LIN {X 0,Y 144.371,Z 167.125,A -85,B 0,C 180,E1 -25963.188,E2 -25963.188} C_VEL
LIN {X 0,Y 141.893,Z 203.573,A -85,B 0,C 180,E1 -25964.823,E2 -25964.823} C_VEL
LIN {X 0,Y 140.005,Z 216.883,A -85,B 0,C 180,E1 -25965.852,E2 -25965.852} C_VEL
LIN {X 0,Y 137.437,Z 229.509,A -85,B 0,C 180,E1 -25967.347,E2 -25967.347} C_VEL
LIN {X 0,Y 134.351,Z 240.695,A -85,B 0,C 180,E1 -25969.164,E2 -25969.164} C_VEL
LIN {X 0,Y 130.518,Z 252.344,A -85,B 0,C 180,E1 -25971.739,E2 -25971.739} C_VEL
LIN {X 0,Y 127.001,Z 261.752,A -85,B 0,C 180,E1 -25974.475,E2 -25974.475} C_VEL
LIN {X 0,Y 123.23,Z 271.427,A -85,B 0,C 180,E1 -25978.16,E2 -25978.16} C_VEL
LIN {X 0,Y 119.16,Z 280.685,A -85,B 0,C 180,E1 -25982.8,E2 -25982.8} C_VEL
LIN {X 0,Y 116.327,Z 288.174,A -85,B 0,C 180,E1 -25987.814,E2 -25987.814} C_VEL
LIN {X 0,Y 113.848,Z 295.01,A -85,B 0,C 180,E1 -25993.871,E2 -25993.871} C_VEL
LIN {X 0,Y 112.764,Z 299.516,A -85,B 0,C 180,E1 -25999.223,E2 -25999.223} C_VEL
LIN {X 0,Y 112.489,Z 301.887,A -85,B 0,C 180,E1 -26002.822,E2 -26002.822} C_VEL
LIN {X 0,Y 112.546,Z 304.345,A -85,B 0,C 180,E1 -26007.618,E2 -26007.618} C_VEL
LIN {X 0,Y 112.706,Z 305.282,A -85,B 0,C 180,E1 -26010,E2 -26010} C_VEL
LIN {X 0,Y 112.583,Z 306.265,A -85,B 0,C 180,E1 -26013.579,E2 -26013.579} C_VEL
LIN {X 0,Y 112.745,Z 307.033,A -85,B 0,C 180,E1 -26020.778,E2 -26020.778} C_VEL
LIN {X 0,Y 113.483,Z 306.842,A -85,B 0,C 180,E1 -26024.342,E2 -26024.342} C_VEL
LIN {X 0,Y 116.179,Z 305.24,A -85,B 0,C 180,E1 -26031.282,E2 -26031.282} C_VEL
LIN {X 0,Y 120.646,Z 302.091,A -85,B 0,C 180,E1 -26037.777,E2 -26037.777} C_VEL
LIN {X 0,Y 125.355,Z 298.158,A -85,B 0,C 180,E1 -26042.757,E2 -26042.757} C_VEL
LIN {X 0,Y 131.716,Z 292.195,A -85,B 0,C 180,E1 -26047.851,E2 -26047.851} C_VEL
LIN {X 0,Y 137.718,Z 286.001,A -85,B 0,C 180,E1 -26051.561,E2 -26051.561} C_VEL
LIN {X 0,Y 144.339,Z 278.329,A -85,B 0,C 180,E1 -26054.912,E2 -26054.912} C_VEL
LIN {X 0,Y 150.335,Z 270.296,A -85,B 0,C 180,E1 -26057.534,E2 -26057.534} C_VEL
LIN {X 0,Y 151.733,Z 267.559,A -85,B 0,C 180,E1 -26058.493,E2 -26058.493} C_VEL
LIN {X 0,Y 154.006,Z 258.604,A -85,B 0,C 180,E1 -26062.192,E2 -26062.192} C_VEL
LIN {X 0,Y 155.453,Z 255.513,A -85,B 0,C 180,E1 -26062.952,E2 -26062.952} C_VEL
LIN {X 0,Y 160.707,Z 245.469,A -85,B 0,C 180,E1 -26064.539,E2 -26064.539} C_VEL
LIN {X 0,Y 165.609,Z 234.176,A -85,B 0,C 180,E1 -26065.846,E2 -26065.846} C_VEL
LIN {X 0,Y 169.472,Z 222.762,A -85,B 0,C 180,E1 -26066.825,E2 -26066.825} C_VEL
LIN {X 0,Y 172.698,Z 209.662,A -85,B 0,C 180,E1 -26067.587,E2 -26067.587} C_VEL
LIN {X 0,Y 174.718,Z 195.983,A -85,B 0,C 180,E1 -26068.133,E2 -26068.133} C_VEL
LIN {X 0,Y 175.367,Z 187.979,A -85,B 0,C 180,E1 -26068.433,E2 -26068.433} C_VEL
LIN {X 0,Y 172.36,Z 179.063,A -85,B 0,C 180,E1 -26071.315,E2 -26071.315} C_VEL
LIN {X 0,Y 169.405,Z 171.309,A -85,B 0,C 180,E1 -26074.505,E2 -26074.505} C_VEL
LIN {X 0,Y 167.011,Z 165.673,A -85,B 0,C 180,E1 -26077.488,E2 -26077.488} C_VEL
LIN {X 0,Y 165.43,Z 161.949,A -85,B 0,C 180,E1 -26079.827,E2 -26079.827} C_VEL
LIN {X 0,Y 163.63,Z 157.962,A -85,B 0,C 180,E1 -26083.037,E2 -26083.037} C_VEL
LIN {X 0,Y 161.693,Z 154.386,A -85,B 0,C 180,E1 -26087.76,E2 -26087.76} C_VEL
LIN {X 0,Y 161.427,Z 153.804,A -85,B 0,C 180,E1 -26088.701,E2 -26088.701} C_VEL
LIN {X 0,Y 160.411,Z 152.94,A -85,B 0,C 180,E1 -26094.973,E2 -26094.973} C_VEL
LIN {X 0,Y 160.784,Z 152.96,A -85,B 0,C 180,E1 -26099.264,E2 -26099.264} C_VEL
LIN {X 0,Y 161.714,Z 154.006,A -85,B 0,C 180,E1 -26102.958,E2 -26102.958} C_VEL
LIN {X 0,Y 163.636,Z 157.763,A -85,B 0,C 180,E1 -26107.713,E2 -26107.713} C_VEL
LIN {X 0,Y 166.289,Z 162.414,A -85,B 0,C 180,E1 -26112.045,E2 -26112.045} C_VEL
LIN {X 0,Y 168.725,Z 166.769,A -85,B 0,C 180,E1 -26115.128,E2 -26115.128} C_VEL
LIN {X 0,Y 171.773,Z 172.259,A -85,B 0,C 180,E1 -26118.332,E2 -26118.332} C_VEL
LIN {X 0,Y 175.556,Z 179.968,A -85,B 0,C 180,E1 -26121.759,E2 -26121.759} C_VEL
LIN {X 0,Y 175.996,Z 180.975,A -85,B 0,C 180,E1 -26122.132,E2 -26122.132} C_VEL
LIN {X 0,Y 174.142,Z 197.162,A -85,B 0,C 180,E1 -26122.723,E2 -26122.723} C_VEL
LIN {X 0,Y 171.684,Z 209.367,A -85,B 0,C 180,E1 -26123.487,E2 -26123.487} C_VEL
LIN {X 0,Y 168.004,Z 222.113,A -85,B 0,C 180,E1 -26124.651,E2 -26124.651} C_VEL
LIN {X 0,Y 163.378,Z 234.084,A -85,B 0,C 180,E1 -26126.106,E2 -26126.106} C_VEL
LIN {X 0,Y 158.006,Z 244.981,A -85,B 0,C 180,E1 -26127.868,E2 -26127.868} C_VEL
LIN {X 0,Y 152.16,Z 254.847,A -85,B 0,C 180,E1 -26129.999,E2 -26129.999} C_VEL
LIN {X 0,Y 146.008,Z 263.789,A -85,B 0,C 180,E1 -26132.61,E2 -26132.61} C_VEL
LIN {X 0,Y 140.002,Z 271.114,A -85,B 0,C 180,E1 -26135.339,E2 -26135.339} C_VEL
LIN {X 0,Y 134.415,Z 277.166,A -85,B 0,C 180,E1 -26138.345,E2 -26138.345} C_VEL
LIN {X 0,Y 128.196,Z 283.07,A -85,B 0,C 180,E1 -26142.26,E2 -26142.26} C_VEL
LIN {X 0,Y 122.548,Z 287.68,A -85,B 0,C 180,E1 -26146.513,E2 -26146.513} C_VEL
LIN {X 0,Y 118.025,Z 290.872,A -85,B 0,C 180,E1 -26150.724,E2 -26150.724} C_VEL
LIN {X 0,Y 113.464,Z 293.574,A -85,B 0,C 180,E1 -26156.119,E2 -26156.119} C_VEL
LIN {X 0,Y 111.17,Z 294.645,A -85,B 0,C 180,E1 -26159.619,E2 -26159.619} C_VEL
LIN {X 0,Y 107.735,Z 295.552,A -85,B 0,C 180,E1 -26166.958,E2 -26166.958} C_VEL
LIN {X 0,Y 106.539,Z 295.422,A -85,B 0,C 180,E1 -26170.741,E2 -26170.741} C_VEL
LIN {X 0,Y 105.734,Z 294.852,A -85,B 0,C 180,E1 -26174.581,E2 -26174.581} C_VEL
LIN {X 0,Y 105.388,Z 293.878,A -85,B 0,C 180,E1 -26178.46,E2 -26178.46} C_VEL
LIN {X 0,Y 105.77,Z 291.147,A -85,B 0,C 180,E1 -26185.332,E2 -26185.332} C_VEL
LIN {X 0,Y 106.744,Z 287.22,A -85,B 0,C 180,E1 -26191.887,E2 -26191.887} C_VEL
LIN {X 0,Y 108.52,Z 282.62,A -85,B 0,C 180,E1 -26197.442,E2 -26197.442} C_VEL
LIN {X 0,Y 111.491,Z 275.685,A -85,B 0,C 180,E1 -26203.674,E2 -26203.674} C_VEL
LIN {X 0,Y 115.036,Z 268.172,A -85,B 0,C 180,E1 -26208.708,E2 -26208.708} C_VEL
LIN {X 0,Y 118.414,Z 260.521,A -85,B 0,C 180,E1 -26212.693,E2 -26212.693} C_VEL
LIN {X 0,Y 122.438,Z 251.174,A -85,B 0,C 180,E1 -26216.415,E2 -26216.415} C_VEL
LIN {X 0,Y 126.508,Z 240.767,A -85,B 0,C 180,E1 -26219.541,E2 -26219.541} C_VEL
LIN {X 0,Y 130.298,Z 229.231,A -85,B 0,C 180,E1 -26222.184,E2 -26222.184} C_VEL
LIN {X 0,Y 133.405,Z 217.085,A -85,B 0,C 180,E1 -26224.267,E2 -26224.267} C_VEL
LIN {X 0,Y 135.877,Z 203.674,A -85,B 0,C 180,E1 -26225.918,E2 -26225.918} C_VEL
LIN {X 0,Y 137.458,Z 190.843,A -85,B 0,C 180,E1 -26226.941,E2 -26226.941} C_VEL
LIN {X 0,Y 140.322,Z 149.589,A -85,B 0,C 180,E1 -26228.789,E2 -26228.789} C_VEL
LIN {X 0,Y 135.901,Z 140.06,A -85,B 0,C 180,E1 -26231.373,E2 -26231.373} C_VEL
LIN {X 0,Y 131.262,Z 131.57,A -85,B 0,C 180,E1 -26234.301,E2 -26234.301} C_VEL
LIN {X 0,Y 126.15,Z 123.395,A -85,B 0,C 180,E1 -26237.916,E2 -26237.916} C_VEL
LIN {X 0,Y 122.463,Z 118.286,A -85,B 0,C 180,E1 -26240.856,E2 -26240.856} C_VEL
LIN {X 0,Y 120.026,Z 114.83,A -85,B 0,C 180,E1 -26243.049,E2 -26243.049} C_VEL
LIN {X 0,Y 117.541,Z 111.714,A -85,B 0,C 180,E1 -26245.488,E2 -26245.488} C_VEL
LIN {X 0,Y 116.829,Z 110.266,A -85,B 0,C 180,E1 -26246.312,E2 -26246.312} C_VEL
LIN {X 0,Y 114.195,Z 107.957,A -85,B 0,C 180,E1 -26249.228,E2 -26249.228} C_VEL
LIN {X 0,Y 112.545,Z 104.889,A -85,B 0,C 180,E1 -26251.566,E2 -26251.566} C_VEL
LIN {X 0,Y 109.927,Z 103.24,A -85,B 0,C 180,E1 -26255.365,E2 -26255.365} C_VEL
LIN {X 0,Y 108.274,Z 100.512,A -85,B 0,C 180,E1 -26258.711,E2 -26258.711} C_VEL
LIN {X 0,Y 107.884,Z 99.025,A -85,B 0,C 180,E1 -26260.001,E2 -26260.001} C_VEL
LIN {X 0,Y 108.177,Z 98.985,A -85,B 0,C 180,E1 -26267.039,E2 -26267.039} C_VEL
LIN {X 0,Y 108.305,Z 98.962,A -85,B 0,C 180,E1 -26272.543,E2 -26272.543} C_VEL
LIN {X 0,Y 108.92,Z 98.908,A -85,B 0,C 180,E1 -26280,E2 -26280} C_VEL
LIN {X 0,Y 108.27,Z 99.01,A -85,B 0,C 180,E1 -26290.165,E2 -26290.165} C_VEL
LIN {X 0,Y 108.973,Z 101.41,A -85,B 0,C 180,E1 -26291.986,E2 -26291.986} C_VEL
LIN {X 0,Y 110.885,Z 103.905,A -85,B 0,C 180,E1 -26295.392,E2 -26295.392} C_VEL
LIN {X 0,Y 112.887,Z 105.114,A -85,B 0,C 180,E1 -26298.137,E2 -26298.137} C_VEL
LIN {X 0,Y 114.533,Z 108.231,A -85,B 0,C 180,E1 -26300.426,E2 -26300.426} C_VEL
LIN {X 0,Y 117.047,Z 110.636,A -85,B 0,C 180,E1 -26303.189,E2 -26303.189} C_VEL
LIN {X 0,Y 119.289,Z 114.04,A -85,B 0,C 180,E1 -26305.52,E2 -26305.52} C_VEL
LIN {X 0,Y 120.811,Z 115.735,A -85,B 0,C 180,E1 -26306.908,E2 -26306.908} C_VEL
LIN {X 0,Y 124.326,Z 120.81,A -85,B 0,C 180,E1 -26309.92,E2 -26309.92} C_VEL
LIN {X 0,Y 128.722,Z 127.364,A -85,B 0,C 180,E1 -26313.209,E2 -26313.209} C_VEL
LIN {X 0,Y 132.754,Z 136.18,A -85,B 0,C 180,E1 -26316.083,E2 -26316.083} C_VEL
LIN {X 0,Y 136.377,Z 145.541,A -85,B 0,C 180,E1 -26318.505,E2 -26318.505} C_VEL
LIN {X 0,Y 138.617,Z 152.722,A -85,B 0,C 180,E1 -26319.99,E2 -26319.99} C_VEL
LIN {X 0,Y 139.093,Z 168.621,A -85,B 0,C 180,E1 -26321.313,E2 -26321.313} C_VEL
LIN {X 0,Y 136.557,Z 203.434,A -85,B 0,C 180,E1 -26322.9,E2 -26322.9} C_VEL
LIN {X 0,Y 134.553,Z 216.833,A -85,B 0,C 180,E1 -26323.959,E2 -26323.959} C_VEL
LIN {X 0,Y 132.023,Z 228.822,A -85,B 0,C 180,E1 -26325.41,E2 -26325.41} C_VEL
LIN {X 0,Y 128.519,Z 240.886,A -85,B 0,C 180,E1 -26327.411,E2 -26327.411} C_VEL
LIN {X 0,Y 124.509,Z 252.43,A -85,B 0,C 180,E1 -26330.053,E2 -26330.053} C_VEL
LIN {X 0,Y 120.805,Z 261.755,A -85,B 0,C 180,E1 -26332.873,E2 -26332.873} C_VEL
LIN {X 0,Y 117.188,Z 270.462,A -85,B 0,C 180,E1 -26336.306,E2 -26336.306} C_VEL
LIN {X 0,Y 114.298,Z 276.8,A -85,B 0,C 180,E1 -26339.411,E2 -26339.411} C_VEL
LIN {X 0,Y 112.238,Z 281.288,A -85,B 0,C 180,E1 -26342.026,E2 -26342.026} C_VEL
LIN {X 0,Y 109.277,Z 288.558,A -85,B 0,C 180,E1 -26347.301,E2 -26347.301} C_VEL
LIN {X 0,Y 106.988,Z 294.362,A -85,B 0,C 180,E1 -26352.806,E2 -26352.806} C_VEL
LIN {X 0,Y 105.766,Z 298.93,A -85,B 0,C 180,E1 -26358.501,E2 -26358.501} C_VEL
LIN {X 0,Y 105.42,Z 301.33,A -85,B 0,C 180,E1 -26362.337,E2 -26362.337} C_VEL
LIN {X 0,Y 105.48,Z 304.085,A -85,B 0,C 180,E1 -26368.092,E2 -26368.092} C_VEL
LIN {X 0,Y 105.608,Z 304.802,A -85,B 0,C 180,E1 -26370,E2 -26370} C_VEL
LIN {X 0,Y 105.495,Z 305.815,A -85,B 0,C 180,E1 -26373.82,E2 -26373.82} C_VEL
LIN {X 0,Y 105.759,Z 306.634,A -85,B 0,C 180,E1 -26381.499,E2 -26381.499} C_VEL
LIN {X 0,Y 106.57,Z 306.478,A -85,B 0,C 180,E1 -26385.295,E2 -26385.295} C_VEL
LIN {X 0,Y 107.8,Z 305.906,A -85,B 0,C 180,E1 -26389.024,E2 -26389.024} C_VEL
LIN {X 0,Y 111.781,Z 303.597,A -85,B 0,C 180,E1 -26396.111,E2 -26396.111} C_VEL
LIN {X 0,Y 115.858,Z 300.796,A -85,B 0,C 180,E1 -26401.039,E2 -26401.039} C_VEL
LIN {X 0,Y 120.643,Z 296.997,A -85,B 0,C 180,E1 -26405.63,E2 -26405.63} C_VEL
LIN {X 0,Y 126.173,Z 292.108,A -85,B 0,C 180,E1 -26409.834,E2 -26409.834} C_VEL
LIN {X 0,Y 132.494,Z 285.984,A -85,B 0,C 180,E1 -26413.596,E2 -26413.596} C_VEL
LIN {X 0,Y 139.397,Z 278.403,A -85,B 0,C 180,E1 -26416.975,E2 -26416.975} C_VEL
LIN {X 0,Y 145.489,Z 270.684,A -85,B 0,C 180,E1 -26419.537,E2 -26419.537} C_VEL
LIN {X 0,Y 152.555,Z 260.232,A -85,B 0,C 180,E1 -26422.086,E2 -26422.086} C_VEL
LIN {X 0,Y 155.453,Z 255.513,A -85,B 0,C 180,E1 -26422.952,E2 -26422.952} C_VEL
LIN {X 0,Y 157.735,Z 250.79,A -85,B 0,C 180,E1 -26423.931,E2 -26423.931} C_VEL
LIN {X 0,Y 160.132,Z 242.902,A -85,B 0,C 180,E1 -26425.914,E2 -26425.914} C_VEL
LIN {X 0,Y 162.217,Z 234.678,A -85,B 0,C 180,E1 -26427.726,E2 -26427.726} C_VEL
LIN {X 0,Y 163.888,Z 229.337,A -85,B 0,C 180,E1 -26428.437,E2 -26428.437} C_VEL
LIN {X 0,Y 167.933,Z 216.125,A -85,B 0,C 180,E1 -26429.373,E2 -26429.373} C_VEL
LIN {X 0,Y 170.635,Z 203.005,A -85,B 0,C 180,E1 -26429.982,E2 -26429.982} C_VEL
LIN {X 0,Y 171.993,Z 190.995,A -85,B 0,C 180,E1 -26430.412,E2 -26430.412} C_VEL
LIN {X 0,Y 169.101,Z 182.07,A -85,B 0,C 180,E1 -26433.545,E2 -26433.545} C_VEL
LIN {X 0,Y 166.5,Z 174.975,A -85,B 0,C 180,E1 -26436.771,E2 -26436.771} C_VEL
LIN {X 0,Y 163.949,Z 168.443,A -85,B 0,C 180,E1 -26440.657,E2 -26440.657} C_VEL
LIN {X 0,Y 162.391,Z 164.745,A -85,B 0,C 180,E1 -26443.661,E2 -26443.661} C_VEL
LIN {X 0,Y 160.595,Z 161.098,A -85,B 0,C 180,E1 -26448.479,E2 -26448.479} C_VEL
LIN {X 0,Y 159.74,Z 160.172,A -85,B 0,C 180,E1 -26452.415,E2 -26452.415} C_VEL
LIN {X 0,Y 159.823,Z 159.956,A -85,B 0,C 180,E1 -26458.74,E2 -26458.74} C_VEL
LIN {X 0,Y 160.683,Z 160.956,A -85,B 0,C 180,E1 -26462.507,E2 -26462.507} C_VEL
LIN {X 0,Y 162.454,Z 164.606,A -85,B 0,C 180,E1 -26467.196,E2 -26467.196} C_VEL
LIN {X 0,Y 164.873,Z 169.197,A -85,B 0,C 180,E1 -26471.407,E2 -26471.407} C_VEL
LIN {X 0,Y 167.262,Z 173.689,A -85,B 0,C 180,E1 -26474.602,E2 -26474.602} C_VEL
LIN {X 0,Y 169.943,Z 178.878,A -85,B 0,C 180,E1 -26477.583,E2 -26477.583} C_VEL
LIN {X 0,Y 172.573,Z 184.626,A -85,B 0,C 180,E1 -26480.168,E2 -26480.168} C_VEL
LIN {X 0,Y 170.743,Z 198.637,A -85,B 0,C 180,E1 -26480.681,E2 -26480.681} C_VEL
LIN {X 0,Y 167.955,Z 211.364,A -85,B 0,C 180,E1 -26481.495,E2 -26481.495} C_VEL
LIN {X 0,Y 164.109,Z 223.915,A -85,B 0,C 180,E1 -26482.67,E2 -26482.67} C_VEL
LIN {X 0,Y 159.627,Z 234.869,A -85,B 0,C 180,E1 -26483.995,E2 -26483.995} C_VEL
LIN {X 0,Y 154.062,Z 245.674,A -85,B 0,C 180,E1 -26485.715,E2 -26485.715} C_VEL
LIN {X 0,Y 147.811,Z 255.787,A -85,B 0,C 180,E1 -26487.897,E2 -26487.897} C_VEL
LIN {X 0,Y 140.957,Z 265.198,A -85,B 0,C 180,E1 -26490.675,E2 -26490.675} C_VEL
LIN {X 0,Y 133.525,Z 273.587,A -85,B 0,C 180,E1 -26494.005,E2 -26494.005} C_VEL
LIN {X 0,Y 127.127,Z 279.857,A -85,B 0,C 180,E1 -26497.453,E2 -26497.453} C_VEL
LIN {X 0,Y 121.328,Z 284.805,A -85,B 0,C 180,E1 -26501.146,E2 -26501.146} C_VEL
LIN {X 0,Y 115.517,Z 289.09,A -85,B 0,C 180,E1 -26505.601,E2 -26505.601} C_VEL
LIN {X 0,Y 110.436,Z 292.27,A -85,B 0,C 180,E1 -26510.477,E2 -26510.477} C_VEL
LIN {X 0,Y 107.498,Z 293.83,A -85,B 0,C 180,E1 -26513.956,E2 -26513.956} C_VEL
LIN {X 0,Y 104.965,Z 294.961,A -85,B 0,C 180,E1 -26517.612,E2 -26517.612} C_VEL
LIN {X 0,Y 101.108,Z 295.929,A -85,B 0,C 180,E1 -26525.351,E2 -26525.351} C_VEL
LIN {X 0,Y 99.757,Z 295.83,A -85,B 0,C 180,E1 -26529.375,E2 -26529.375} C_VEL
LIN {X 0,Y 98.793,Z 295.319,A -85,B 0,C 180,E1 -26533.468,E2 -26533.468} C_VEL
LIN {X 0,Y 98.339,Z 294.374,A -85,B 0,C 180,E1 -26537.62,E2 -26537.62} C_VEL
LIN {X 0,Y 98.695,Z 291.476,A -85,B 0,C 180,E1 -26545.503,E2 -26545.503} C_VEL
LIN {X 0,Y 99.646,Z 287.846,A -85,B 0,C 180,E1 -26552.021,E2 -26552.021} C_VEL
LIN {X 0,Y 101.497,Z 283.321,A -85,B 0,C 180,E1 -26557.961,E2 -26557.961} C_VEL
LIN {X 0,Y 104.605,Z 276.484,A -85,B 0,C 180,E1 -26564.593,E2 -26564.593} C_VEL
LIN {X 0,Y 108.356,Z 269.056,A -85,B 0,C 180,E1 -26569.909,E2 -26569.909} C_VEL
LIN {X 0,Y 111.934,Z 261.504,A -85,B 0,C 180,E1 -26574.087,E2 -26574.087} C_VEL
LIN {X 0,Y 116.138,Z 252.336,A -85,B 0,C 180,E1 -26577.969,E2 -26577.969} C_VEL
LIN {X 0,Y 120.38,Z 242.112,A -85,B 0,C 180,E1 -26581.208,E2 -26581.208} C_VEL
LIN {X 0,Y 124.385,Z 230.781,A -85,B 0,C 180,E1 -26583.915,E2 -26583.915} C_VEL
LIN {X 0,Y 127.667,Z 219.064,A -85,B 0,C 180,E1 -26586.04,E2 -26586.04} C_VEL
LIN {X 0,Y 130.268,Z 206.292,A -85,B 0,C 180,E1 -26587.726,E2 -26587.726} C_VEL
LIN {X 0,Y 132.135,Z 192.787,A -85,B 0,C 180,E1 -26588.898,E2 -26588.898} C_VEL
LIN {X 0,Y 135.181,Z 151.945,A -85,B 0,C 180,E1 -26590.79,E2 -26590.79} C_VEL
LIN {X 0,Y 131.121,Z 143.155,A -85,B 0,C 180,E1 -26593.409,E2 -26593.409} C_VEL
LIN {X 0,Y 126.794,Z 135.129,A -85,B 0,C 180,E1 -26596.443,E2 -26596.443} C_VEL
LIN {X 0,Y 122.314,Z 127.979,A -85,B 0,C 180,E1 -26599.955,E2 -26599.955} C_VEL
LIN {X 0,Y 119.3,Z 123.587,A -85,B 0,C 180,E1 -26602.625,E2 -26602.625} C_VEL
LIN {X 0,Y 117.486,Z 120.881,A -85,B 0,C 180,E1 -26604.413,E2 -26604.413} C_VEL
LIN {X 0,Y 114.951,Z 117.413,A -85,B 0,C 180,E1 -26607.142,E2 -26607.142} C_VEL
LIN {X 0,Y 114.18,Z 116.359,A -85,B 0,C 180,E1 -26608.049,E2 -26608.049} C_VEL
LIN {X 0,Y 111.847,Z 113.755,A -85,B 0,C 180,E1 -26610.978,E2 -26610.978} C_VEL
LIN {X 0,Y 110.772,Z 111.622,A -85,B 0,C 180,E1 -26612.655,E2 -26612.655} C_VEL
LIN {X 0,Y 108.173,Z 109.622,A -85,B 0,C 180,E1 -26616.819,E2 -26616.819} C_VEL
LIN {X 0,Y 106.685,Z 106.794,A -85,B 0,C 180,E1 -26620.269,E2 -26620.269} C_VEL
LIN {X 0,Y 106.364,Z 105.942,A -85,B 0,C 180,E1 -26621.21,E2 -26621.21} C_VEL
LIN {X 0,Y 103.763,Z 104.443,A -85,B 0,C 180,E1 -26632.215,E2 -26632.215} C_VEL
LIN {X 0,Y 104.224,Z 104.336,A -85,B 0,C 180,E1 -26640.483,E2 -26640.483} C_VEL
LIN {X 0,Y 106.798,Z 106.137,A -85,B 0,C 180,E1 -26649.042,E2 -26649.042} C_VEL
LIN {X 0,Y 108.097,Z 109.161,A -85,B 0,C 180,E1 -26652.199,E2 -26652.199} C_VEL
LIN {X 0,Y 110.242,Z 111.258,A -85,B 0,C 180,E1 -26655.839,E2 -26655.839} C_VEL
LIN {X 0,Y 111.072,Z 111.982,A -85,B 0,C 180,E1 -26657.046,E2 -26657.046} C_VEL
LIN {X 0,Y 112.976,Z 115.135,A -85,B 0,C 180,E1 -26659.771,E2 -26659.771} C_VEL
LIN {X 0,Y 114.795,Z 116.994,A -85,B 0,C 180,E1 -26661.906,E2 -26661.906} C_VEL
LIN {X 0,Y 117.423,Z 120.762,A -85,B 0,C 180,E1 -26664.77,E2 -26664.77} C_VEL
LIN {X 0,Y 121.111,Z 126.062,A -85,B 0,C 180,E1 -26668.249,E2 -26668.249} C_VEL
LIN {X 0,Y 125.451,Z 132.911,A -85,B 0,C 180,E1 -26671.801,E2 -26671.801} C_VEL
LIN {X 0,Y 129.768,Z 143.114,A -85,B 0,C 180,E1 -26675.14,E2 -26675.14} C_VEL
LIN {X 0,Y 133.589,Z 154.367,A -85,B 0,C 180,E1 -26677.923,E2 -26677.923} C_VEL
LIN {X 0,Y 134.045,Z 168.599,A -85,B 0,C 180,E1 -26679.218,E2 -26679.218} C_VEL
LIN {X 0,Y 131.514,Z 202.469,A -85,B 0,C 180,E1 -26680.791,E2 -26680.791} C_VEL
LIN {X 0,Y 129.435,Z 215.975,A -85,B 0,C 180,E1 -26681.849,E2 -26681.849} C_VEL
LIN {X 0,Y 126.773,Z 228.088,A -85,B 0,C 180,E1 -26683.312,E2 -26683.312} C_VEL
LIN {X 0,Y 123.382,Z 239.46,A -85,B 0,C 180,E1 -26685.178,E2 -26685.178} C_VEL
LIN {X 0,Y 120.222,Z 248.562,A -85,B 0,C 180,E1 -26687.188,E2 -26687.188} C_VEL
LIN {X 0,Y 115.58,Z 259.567,A -85,B 0,C 180,E1 -26690.322,E2 -26690.322} C_VEL
LIN {X 0,Y 112.112,Z 267.679,A -85,B 0,C 180,E1 -26693.449,E2 -26693.449} C_VEL
LIN {X 0,Y 108.084,Z 276.238,A -85,B 0,C 180,E1 -26697.669,E2 -26697.669} C_VEL
LIN {X 0,Y 105.753,Z 280.839,A -85,B 0,C 180,E1 -26700.45,E2 -26700.45} C_VEL
LIN {X 0,Y 102.709,Z 287.81,A -85,B 0,C 180,E1 -26705.76,E2 -26705.76} C_VEL
LIN {X 0,Y 100.181,Z 293.703,A -85,B 0,C 180,E1 -26711.597,E2 -26711.597} C_VEL
LIN {X 0,Y 98.759,Z 298.338,A -85,B 0,C 180,E1 -26717.673,E2 -26717.673} C_VEL
LIN {X 0,Y 98.347,Z 300.772,A -85,B 0,C 180,E1 -26721.783,E2 -26721.783} C_VEL
LIN {X 0,Y 98.431,Z 303.75,A -85,B 0,C 180,E1 -26728.416,E2 -26728.416} C_VEL
LIN {X 0,Y 98.445,Z 304.824,A -85,B 0,C 180,E1 -26731.86,E2 -26731.86} C_VEL
LIN {X 0,Y 98.349,Z 305.988,A -85,B 0,C 180,E1 -26738.217,E2 -26738.217} C_VEL
LIN {X 0,Y 99.7,Z 306.104,A -85,B 0,C 180,E1 -26746.377,E2 -26746.377} C_VEL
LIN {X 0,Y 101.079,Z 305.584,A -85,B 0,C 180,E1 -26750.343,E2 -26750.343} C_VEL
LIN {X 0,Y 105.418,Z 303.33,A -85,B 0,C 180,E1 -26757.819,E2 -26757.819} C_VEL
LIN {X 0,Y 109.803,Z 300.585,A -85,B 0,C 180,E1 -26762.96,E2 -26762.96} C_VEL
LIN {X 0,Y 114.932,Z 296.846,A -85,B 0,C 180,E1 -26767.698,E2 -26767.698} C_VEL
LIN {X 0,Y 120.806,Z 292.021,A -85,B 0,C 180,E1 -26771.992,E2 -26771.992} C_VEL
LIN {X 0,Y 127.445,Z 285.967,A -85,B 0,C 180,E1 -26775.798,E2 -26775.798} C_VEL
LIN {X 0,Y 134.65,Z 278.465,A -85,B 0,C 180,E1 -26779.185,E2 -26779.185} C_VEL
LIN {X 0,Y 140.99,Z 270.837,A -85,B 0,C 180,E1 -26781.73,E2 -26781.73} C_VEL
LIN {X 0,Y 147.612,Z 261.615,A -85,B 0,C 180,E1 -26784.037,E2 -26784.037} C_VEL
LIN {X 0,Y 153.194,Z 252.645,A -85,B 0,C 180,E1 -26785.668,E2 -26785.668} C_VEL
LIN {X 0,Y 158.865,Z 241.602,A -85,B 0,C 180,E1 -26787.197,E2 -26787.197} C_VEL
LIN {X 0,Y 163.888,Z 229.337,A -85,B 0,C 180,E1 -26788.437,E2 -26788.437} C_VEL
LIN {X 0,Y 164.842,Z 225.742,A -85,B 0,C 180,E1 -26788.951,E2 -26788.951} C_VEL
LIN {X 0,Y 165.341,Z 220.112,A -85,B 0,C 180,E1 -26790.25,E2 -26790.25} C_VEL
LIN {X 0,Y 165.642,Z 214.358,A -85,B 0,C 180,E1 -26791.465,E2 -26791.465} C_VEL
LIN {X 0,Y 166.219,Z 210.576,A -85,B 0,C 180,E1 -26791.843,E2 -26791.843} C_VEL
LIN {X 0,Y 168.391,Z 197.785,A -85,B 0,C 180,E1 -26792.355,E2 -26792.355} C_VEL
LIN {X 0,Y 168.795,Z 194.083,A -85,B 0,C 180,E1 -26792.488,E2 -26792.488} C_VEL
LIN {X 0,Y 166.577,Z 186.757,A -85,B 0,C 180,E1 -26795.211,E2 -26795.211} C_VEL
LIN {X 0,Y 164.431,Z 180.436,A -85,B 0,C 180,E1 -26798.203,E2 -26798.203} C_VEL
LIN {X 0,Y 162.329,Z 174.605,A -85,B 0,C 180,E1 -26801.811,E2 -26801.811} C_VEL
LIN {X 0,Y 161.081,Z 171.394,A -85,B 0,C 180,E1 -26804.49,E2 -26804.49} C_VEL
LIN {X 0,Y 159.523,Z 167.814,A -85,B 0,C 180,E1 -26809.208,E2 -26809.208} C_VEL
LIN {X 0,Y 158.671,Z 167.039,A -85,B 0,C 180,E1 -26814.917,E2 -26814.917} C_VEL
LIN {X 0,Y 158.949,Z 167.008,A -85,B 0,C 180,E1 -26818.733,E2 -26818.733} C_VEL
LIN {X 0,Y 159.657,Z 167.938,A -85,B 0,C 180,E1 -26822.049,E2 -26822.049} C_VEL
LIN {X 0,Y 161.587,Z 172.161,A -85,B 0,C 180,E1 -26827.34,E2 -26827.34} C_VEL
LIN {X 0,Y 163.624,Z 176.25,A -85,B 0,C 180,E1 -26830.988,E2 -26830.988} C_VEL
LIN {X 0,Y 166.198,Z 181.331,A -85,B 0,C 180,E1 -26834.541,E2 -26834.541} C_VEL
LIN {X 0,Y 169.03,Z 187.503,A -85,B 0,C 180,E1 -26837.779,E2 -26837.779} C_VEL
LIN {X 0,Y 169.273,Z 188.079,A -85,B 0,C 180,E1 -26838.046,E2 -26838.046} C_VEL
LIN {X 0,Y 167.298,Z 201.388,A -85,B 0,C 180,E1 -26838.629,E2 -26838.629} C_VEL
LIN {X 0,Y 164.063,Z 214.777,A -85,B 0,C 180,E1 -26839.537,E2 -26839.537} C_VEL
LIN {X 0,Y 159.658,Z 227.45,A -85,B 0,C 180,E1 -26840.766,E2 -26840.766} C_VEL
LIN {X 0,Y 154.646,Z 238.535,A -85,B 0,C 180,E1 -26842.186,E2 -26842.186} C_VEL
LIN {X 0,Y 148.221,Z 249.87,A -85,B 0,C 180,E1 -26844.111,E2 -26844.111} C_VEL
LIN {X 0,Y 141.366,Z 259.881,A -85,B 0,C 180,E1 -26846.508,E2 -26846.508} C_VEL
LIN {X 0,Y 134.741,Z 268.036,A -85,B 0,C 180,E1 -26849.112,E2 -26849.112} C_VEL
LIN {X 0,Y 127.136,Z 275.978,A -85,B 0,C 180,E1 -26852.54,E2 -26852.54} C_VEL
LIN {X 0,Y 121.177,Z 281.326,A -85,B 0,C 180,E1 -26855.711,E2 -26855.711} C_VEL
LIN {X 0,Y 114.52,Z 286.499,A -85,B 0,C 180,E1 -26859.904,E2 -26859.904} C_VEL
LIN {X 0,Y 108.516,Z 290.472,A -85,B 0,C 180,E1 -26864.569,E2 -26864.569} C_VEL
LIN {X 0,Y 104.933,Z 292.493,A -85,B 0,C 180,E1 -26867.951,E2 -26867.951} C_VEL
LIN {X 0,Y 101.712,Z 294.085,A -85,B 0,C 180,E1 -26871.547,E2 -26871.547} C_VEL
LIN {X 0,Y 98.896,Z 295.264,A -85,B 0,C 180,E1 -26875.353,E2 -26875.353} C_VEL
LIN {X 0,Y 94.948,Z 296.281,A -85,B 0,C 180,E1 -26882.652,E2 -26882.652} C_VEL
LIN {X 0,Y 93.026,Z 296.236,A -85,B 0,C 180,E1 -26887.806,E2 -26887.806} C_VEL
LIN {X 0,Y 91.895,Z 295.777,A -85,B 0,C 180,E1 -26892.187,E2 -26892.187} C_VEL
LIN {X 0,Y 91.312,Z 294.87,A -85,B 0,C 180,E1 -26896.65,E2 -26896.65} C_VEL
LIN {X 0,Y 91.199,Z 293.561,A -85,B 0,C 180,E1 -26901.134,E2 -26901.134} C_VEL
LIN {X 0,Y 91.729,Z 291.241,A -85,B 0,C 180,E1 -26906.937,E2 -26906.937} C_VEL
LIN {X 0,Y 93.041,Z 287.092,A -85,B 0,C 180,E1 -26914.332,E2 -26914.332} C_VEL
LIN {X 0,Y 95.289,Z 282.25,A -85,B 0,C 180,E1 -26920.626,E2 -26920.626} C_VEL
LIN {X 0,Y 98.352,Z 276.165,A -85,B 0,C 180,E1 -26926.609,E2 -26926.609} C_VEL
LIN {X 0,Y 102.453,Z 268.587,A -85,B 0,C 180,E1 -26932.166,E2 -26932.166} C_VEL
LIN {X 0,Y 106.342,Z 260.855,A -85,B 0,C 180,E1 -26936.494,E2 -26936.494} C_VEL
LIN {X 0,Y 110.898,Z 251.386,A -85,B 0,C 180,E1 -26940.464,E2 -26940.464} C_VEL
LIN {X 0,Y 115.455,Z 240.862,A -85,B 0,C 180,E1 -26943.743,E2 -26943.743} C_VEL
LIN {X 0,Y 119.658,Z 229.161,A -85,B 0,C 180,E1 -26946.491,E2 -26946.491} C_VEL
LIN {X 0,Y 123.108,Z 216.69,A -85,B 0,C 180,E1 -26948.639,E2 -26948.639} C_VEL
LIN {X 0,Y 125.762,Z 203.369,A -85,B 0,C 180,E1 -26950.29,E2 -26950.29} C_VEL
LIN {X 0,Y 127.443,Z 190.212,A -85,B 0,C 180,E1 -26951.309,E2 -26951.309} C_VEL
LIN {X 0,Y 130.186,Z 154.306,A -85,B 0,C 180,E1 -26952.959,E2 -26952.959} C_VEL
LIN {X 0,Y 125.815,Z 144.858,A -85,B 0,C 180,E1 -26956.125,E2 -26956.125} C_VEL
LIN {X 0,Y 121.458,Z 136.997,A -85,B 0,C 180,E1 -26959.615,E2 -26959.615} C_VEL
LIN {X 0,Y 116.909,Z 129.812,A -85,B 0,C 180,E1 -26963.825,E2 -26963.825} C_VEL
LIN {X 0,Y 114.851,Z 126.777,A -85,B 0,C 180,E1 -26966.003,E2 -26966.003} C_VEL
LIN {X 0,Y 112.047,Z 122.723,A -85,B 0,C 180,E1 -26969.373,E2 -26969.373} C_VEL
LIN {X 0,Y 109.654,Z 119.617,A -85,B 0,C 180,E1 -26972.725,E2 -26972.725} C_VEL
LIN {X 0,Y 108.959,Z 118.287,A -85,B 0,C 180,E1 -26973.902,E2 -26973.902} C_VEL
LIN {X 0,Y 106.332,Z 115.729,A -85,B 0,C 180,E1 -26978.684,E2 -26978.684} C_VEL
LIN {X 0,Y 105.144,Z 112.948,A -85,B 0,C 180,E1 -26981.993,E2 -26981.993} C_VEL
LIN {X 0,Y 102.896,Z 111.498,A -85,B 0,C 180,E1 -26992.149,E2 -26992.149} C_VEL
LIN {X 0,Y 103.344,Z 111.429,A -85,B 0,C 180,E1 -27000.488,E2 -27000.488} C_VEL
LIN {X 0,Y 105.416,Z 112.981,A -85,B 0,C 180,E1 -27007.918,E2 -27007.918} C_VEL
LIN {X 0,Y 107.055,Z 116.435,A -85,B 0,C 180,E1 -27012.031,E2 -27012.031} C_VEL
LIN {X 0,Y 109.283,Z 118.644,A -85,B 0,C 180,E1 -27015.862,E2 -27015.862} C_VEL
LIN {X 0,Y 111.484,Z 122.03,A -85,B 0,C 180,E1 -27019.153,E2 -27019.153} C_VEL
LIN {X 0,Y 112.723,Z 123.52,A -85,B 0,C 180,E1 -27020.723,E2 -27020.723} C_VEL
LIN {X 0,Y 116.124,Z 128.548,A -85,B 0,C 180,E1 -27024.607,E2 -27024.607} C_VEL
LIN {X 0,Y 120.265,Z 134.93,A -85,B 0,C 180,E1 -27028.585,E2 -27028.585} C_VEL
LIN {X 0,Y 122.466,Z 138.993,A -85,B 0,C 180,E1 -27030.506,E2 -27030.506} C_VEL
LIN {X 0,Y 126.207,Z 148.587,A -85,B 0,C 180,E1 -27033.682,E2 -27033.682} C_VEL
LIN {X 0,Y 128.936,Z 157.158,A -85,B 0,C 180,E1 -27035.891,E2 -27035.891} C_VEL
LIN {X 0,Y 129.115,Z 169.756,A -85,B 0,C 180,E1 -27037.024,E2 -27037.024} C_VEL
LIN {X 0,Y 126.425,Z 202.871,A -85,B 0,C 180,E1 -27038.579,E2 -27038.579} C_VEL
LIN {X 0,Y 124.157,Z 216.618,A -85,B 0,C 180,E1 -27039.691,E2 -27039.691} C_VEL
LIN {X 0,Y 121.398,Z 228.459,A -85,B 0,C 180,E1 -27041.183,E2 -27041.183} C_VEL
LIN {X 0,Y 117.851,Z 239.618,A -85,B 0,C 180,E1 -27043.069,E2 -27043.069} C_VEL
LIN {X 0,Y 113.997,Z 249.962,A -85,B 0,C 180,E1 -27045.469,E2 -27045.469} C_VEL
LIN {X 0,Y 109.175,Z 260.631,A -85,B 0,C 180,E1 -27048.712,E2 -27048.712} C_VEL
LIN {X 0,Y 104.71,Z 270.314,A -85,B 0,C 180,E1 -27052.837,E2 -27052.837} C_VEL
LIN {X 0,Y 100.328,Z 278.456,A -85,B 0,C 180,E1 -27057.357,E2 -27057.357} C_VEL
LIN {X 0,Y 96.727,Z 285.909,A -85,B 0,C 180,E1 -27062.991,E2 -27062.991} C_VEL
LIN {X 0,Y 94.23,Z 291.18,A -85,B 0,C 180,E1 -27068.104,E2 -27068.104} C_VEL
LIN {X 0,Y 92.207,Z 296.274,A -85,B 0,C 180,E1 -27074.527,E2 -27074.527} C_VEL
LIN {X 0,Y 91.309,Z 300.21,A -85,B 0,C 180,E1 -27081.144,E2 -27081.144} C_VEL
LIN {X 0,Y 91.379,Z 303.481,A -85,B 0,C 180,E1 -27089.009,E2 -27089.009} C_VEL
LIN {X 0,Y 91.297,Z 304.911,A -85,B 0,C 180,E1 -27094.415,E2 -27094.415} C_VEL
LIN {X 0,Y 91.839,Z 305.835,A -85,B 0,C 180,E1 -27103.272,E2 -27103.272} C_VEL
LIN {X 0,Y 94.419,Z 305.25,A -85,B 0,C 180,E1 -27111.849,E2 -27111.849} C_VEL
LIN {X 0,Y 99.163,Z 303.064,A -85,B 0,C 180,E1 -27119.743,E2 -27119.743} C_VEL
LIN {X 0,Y 103.889,Z 300.375,A -85,B 0,C 180,E1 -27125.101,E2 -27125.101} C_VEL
LIN {X 0,Y 109.368,Z 296.695,A -85,B 0,C 180,E1 -27129.986,E2 -27129.986} C_VEL
LIN {X 0,Y 115.612,Z 291.934,A -85,B 0,C 180,E1 -27134.353,E2 -27134.353} C_VEL
LIN {X 0,Y 123.814,Z 284.828,A -85,B 0,C 180,E1 -27138.773,E2 -27138.773} C_VEL
LIN {X 0,Y 131.412,Z 277.157,A -85,B 0,C 180,E1 -27142.077,E2 -27142.077} C_VEL
LIN {X 0,Y 139.453,Z 267.55,A -85,B 0,C 180,E1 -27144.98,E2 -27144.98} C_VEL
LIN {X 0,Y 145.746,Z 258.732,A -85,B 0,C 180,E1 -27146.913,E2 -27146.913} C_VEL
LIN {X 0,Y 152.203,Z 247.964,A -85,B 0,C 180,E1 -27148.676,E2 -27148.676} C_VEL
LIN {X 0,Y 157.376,Z 237.492,A -85,B 0,C 180,E1 -27149.91,E2 -27149.91} C_VEL
LIN {X 0,Y 161.708,Z 226.446,A -85,B 0,C 180,E1 -27150.889,E2 -27150.889} C_VEL
LIN {X 0,Y 165.6,Z 213.146,A -85,B 0,C 180,E1 -27151.723,E2 -27151.723} C_VEL
LIN {X 0,Y 166.219,Z 210.576,A -85,B 0,C 180,E1 -27151.843,E2 -27151.843} C_VEL
LIN {X 0,Y 166.796,Z 206.823,A -85,B 0,C 180,E1 -27152.161,E2 -27152.161} C_VEL
LIN {X 0,Y 166.759,Z 201.609,A -85,B 0,C 180,E1 -27153.119,E2 -27153.119} C_VEL
LIN {X 0,Y 166.002,Z 197.073,A -85,B 0,C 180,E1 -27154.439,E2 -27154.439} C_VEL
LIN {X 0,Y 164.453,Z 191.713,A -85,B 0,C 180,E1 -27156.643,E2 -27156.643} C_VEL
LIN {X 0,Y 162.84,Z 187.037,A -85,B 0,C 180,E1 -27159.057,E2 -27159.057} C_VEL
LIN {X 0,Y 160.889,Z 181.006,A -85,B 0,C 180,E1 -27162.759,E2 -27162.759} C_VEL
LIN {X 0,Y 159.788,Z 177.981,A -85,B 0,C 180,E1 -27165.383,E2 -27165.383} C_VEL
LIN {X 0,Y 158.495,Z 174.747,A -85,B 0,C 180,E1 -27169.783,E2 -27169.783} C_VEL
LIN {X 0,Y 157.919,Z 173.933,A -85,B 0,C 180,E1 -27177.449,E2 -27177.449} C_VEL
LIN {X 0,Y 158.615,Z 174.753,A -85,B 0,C 180,E1 -27181.428,E2 -27181.428} C_VEL
LIN {X 0,Y 160.386,Z 179,A -85,B 0,C 180,E1 -27186.763,E2 -27186.763} C_VEL
LIN {X 0,Y 162.27,Z 183.048,A -85,B 0,C 180,E1 -27190.37,E2 -27190.37} C_VEL
LIN {X 0,Y 164.487,Z 187.801,A -85,B 0,C 180,E1 -27193.67,E2 -27193.67} C_VEL
LIN {X 0,Y 166.212,Z 191.911,A -85,B 0,C 180,E1 -27195.954,E2 -27195.954} C_VEL
LIN {X 0,Y 164.034,Z 204.423,A -85,B 0,C 180,E1 -27196.53,E2 -27196.53} C_VEL
LIN {X 0,Y 160.866,Z 216.255,A -85,B 0,C 180,E1 -27197.341,E2 -27197.341} C_VEL
LIN {X 0,Y 156.609,Z 228.001,A -85,B 0,C 180,E1 -27198.456,E2 -27198.456} C_VEL
LIN {X 0,Y 151.318,Z 239.295,A -85,B 0,C 180,E1 -27199.861,E2 -27199.861} C_VEL
LIN {X 0,Y 145.394,Z 249.433,A -85,B 0,C 180,E1 -27201.487,E2 -27201.487} C_VEL
LIN {X 0,Y 138.272,Z 259.597,A -85,B 0,C 180,E1 -27203.809,E2 -27203.809} C_VEL
LIN {X 0,Y 131.374,Z 267.866,A -85,B 0,C 180,E1 -27206.355,E2 -27206.355} C_VEL
LIN {X 0,Y 123.375,Z 275.923,A -85,B 0,C 180,E1 -27209.691,E2 -27209.691} C_VEL
LIN {X 0,Y 117.065,Z 281.336,A -85,B 0,C 180,E1 -27212.808,E2 -27212.808} C_VEL
LIN {X 0,Y 110.002,Z 286.596,A -85,B 0,C 180,E1 -27217.001,E2 -27217.001} C_VEL
LIN {X 0,Y 103.54,Z 290.644,A -85,B 0,C 180,E1 -27221.699,E2 -27221.699} C_VEL
LIN {X 0,Y 99.662,Z 292.717,A -85,B 0,C 180,E1 -27225.156,E2 -27225.156} C_VEL
LIN {X 0,Y 96.125,Z 294.341,A -85,B 0,C 180,E1 -27228.851,E2 -27228.851} C_VEL
LIN {X 0,Y 93.019,Z 295.551,A -85,B 0,C 180,E1 -27232.812,E2 -27232.812} C_VEL
LIN {X 0,Y 90.344,Z 296.336,A -85,B 0,C 180,E1 -27237.007,E2 -27237.007} C_VEL
LIN {X 0,Y 88.138,Z 296.683,A -85,B 0,C 180,E1 -27241.417,E2 -27241.417} C_VEL
LIN {X 0,Y 86.363,Z 296.643,A -85,B 0,C 180,E1 -27245.991,E2 -27245.991} C_VEL
LIN {X 0,Y 85.051,Z 296.218,A -85,B 0,C 180,E1 -27250.699,E2 -27250.699} C_VEL
LIN {X 0,Y 84.303,Z 295.366,A -85,B 0,C 180,E1 -27255.517,E2 -27255.517} C_VEL
LIN {X 0,Y 84.104,Z 294.086,A -85,B 0,C 180,E1 -27260.38,E2 -27260.38} C_VEL
LIN {X 0,Y 84.545,Z 292.12,A -85,B 0,C 180,E1 -27265.963,E2 -27265.963} C_VEL
LIN {X 0,Y 85.46,Z 289.074,A -85,B 0,C 180,E1 -27272.357,E2 -27272.357} C_VEL
LIN {X 0,Y 87.483,Z 284.686,A -85,B 0,C 180,E1 -27279.246,E2 -27279.246} C_VEL
LIN {X 0,Y 90.368,Z 279.128,A -85,B 0,C 180,E1 -27285.796,E2 -27285.796} C_VEL
LIN {X 0,Y 94.361,Z 272.178,A -85,B 0,C 180,E1 -27291.864,E2 -27291.864} C_VEL
LIN {X 0,Y 99.218,Z 263.468,A -85,B 0,C 180,E1 -27297.415,E2 -27297.415} C_VEL
LIN {X 0,Y 104.326,Z 253.582,A -85,B 0,C 180,E1 -27302.04,E2 -27302.04} C_VEL
LIN {X 0,Y 109.057,Z 243.501,A -85,B 0,C 180,E1 -27305.451,E2 -27305.451} C_VEL
LIN {X 0,Y 113.507,Z 232.305,A -85,B 0,C 180,E1 -27308.256,E2 -27308.256} C_VEL
LIN {X 0,Y 117.435,Z 219.791,A -85,B 0,C 180,E1 -27310.605,E2 -27310.605} C_VEL
LIN {X 0,Y 120.295,Z 207.145,A -85,B 0,C 180,E1 -27312.317,E2 -27312.317} C_VEL
LIN {X 0,Y 122.272,Z 194.325,A -85,B 0,C 180,E1 -27313.476,E2 -27313.476} C_VEL
LIN {X 0,Y 124.754,Z 165.352,A -85,B 0,C 180,E1 -27314.881,E2 -27314.881} C_VEL
LIN {X 0,Y 125.421,Z 156.816,A -85,B 0,C 180,E1 -27315.271,E2 -27315.271} C_VEL
LIN {X 0,Y 121.143,Z 147.578,A -85,B 0,C 180,E1 -27318.754,E2 -27318.754} C_VEL
LIN {X 0,Y 117.037,Z 140.072,A -85,B 0,C 180,E1 -27322.52,E2 -27322.52} C_VEL
LIN {X 0,Y 112.801,Z 133.217,A -85,B 0,C 180,E1 -27327.097,E2 -27327.097} C_VEL
LIN {X 0,Y 109.925,Z 128.977,A -85,B 0,C 180,E1 -27330.824,E2 -27330.824} C_VEL
LIN {X 0,Y 107.583,Z 125.537,A -85,B 0,C 180,E1 -27334.503,E2 -27334.503} C_VEL
LIN {X 0,Y 107.226,Z 124.917,A -85,B 0,C 180,E1 -27335.157,E2 -27335.157} C_VEL
LIN {X 0,Y 104.775,Z 122.118,A -85,B 0,C 180,E1 -27340.172,E2 -27340.172} C_VEL
LIN {X 0,Y 103.787,Z 119.791,A -85,B 0,C 180,E1 -27343.275,E2 -27343.275} C_VEL
LIN {X 0,Y 101.946,Z 118.449,A -85,B 0,C 180,E1 -27354.065,E2 -27354.065} C_VEL
LIN {X 0,Y 102.501,Z 118.595,A -85,B 0,C 180,E1 -27360.737,E2 -27360.737} C_VEL
LIN {X 0,Y 104.157,Z 119.997,A -85,B 0,C 180,E1 -27367.025,E2 -27367.025} C_VEL
LIN {X 0,Y 105.844,Z 123.415,A -85,B 0,C 180,E1 -27371.491,E2 -27371.491} C_VEL
LIN {X 0,Y 107.617,Z 125.346,A -85,B 0,C 180,E1 -27374.756,E2 -27374.756} C_VEL
LIN {X 0,Y 109.919,Z 128.849,A -85,B 0,C 180,E1 -27378.403,E2 -27378.403} C_VEL
LIN {X 0,Y 113.527,Z 134.325,A -85,B 0,C 180,E1 -27383.004,E2 -27383.004} C_VEL
LIN {X 0,Y 117.478,Z 140.787,A -85,B 0,C 180,E1 -27387.155,E2 -27387.155} C_VEL
LIN {X 0,Y 119.14,Z 144.135,A -85,B 0,C 180,E1 -27388.76,E2 -27388.76} C_VEL
LIN {X 0,Y 122.492,Z 153.339,A -85,B 0,C 180,E1 -27391.924,E2 -27391.924} C_VEL
LIN {X 0,Y 124.398,Z 159.84,A -85,B 0,C 180,E1 -27393.668,E2 -27393.668} C_VEL
LIN {X 0,Y 124.368,Z 170.99,A -85,B 0,C 180,E1 -27394.654,E2 -27394.654} C_VEL
LIN {X 0,Y 121.616,Z 202.892,A -85,B 0,C 180,E1 -27396.172,E2 -27396.172} C_VEL
LIN {X 0,Y 119.257,Z 216.51,A -85,B 0,C 180,E1 -27397.289,E2 -27397.289} C_VEL
LIN {X 0,Y 116.191,Z 228.766,A -85,B 0,C 180,E1 -27398.851,E2 -27398.851} C_VEL
LIN {X 0,Y 111.876,Z 241.362,A -85,B 0,C 180,E1 -27401.075,E2 -27401.075} C_VEL
LIN {X 0,Y 107.267,Z 252.612,A -85,B 0,C 180,E1 -27403.886,E2 -27403.886} C_VEL
LIN {X 0,Y 102.916,Z 261.701,A -85,B 0,C 180,E1 -27406.93,E2 -27406.93} C_VEL
LIN {X 0,Y 98.197,Z 271.057,A -85,B 0,C 180,E1 -27411.226,E2 -27411.226} C_VEL
LIN {X 0,Y 93.916,Z 278.399,A -85,B 0,C 180,E1 -27415.557,E2 -27415.557} C_VEL
LIN {X 0,Y 89.797,Z 286.285,A -85,B 0,C 180,E1 -27421.991,E2 -27421.991} C_VEL
LIN {X 0,Y 86.718,Z 292.33,A -85,B 0,C 180,E1 -27428.61,E2 -27428.61} C_VEL
LIN {X 0,Y 84.84,Z 297.099,A -85,B 0,C 180,E1 -27435.61,E2 -27435.61} C_VEL
LIN {X 0,Y 84.129,Z 300.726,A -85,B 0,C 180,E1 -27442.801,E2 -27442.801} C_VEL
LIN {X 0,Y 84.341,Z 303.467,A -85,B 0,C 180,E1 -27450.558,E2 -27450.558} C_VEL
LIN {X 0,Y 84.203,Z 304.445,A -85,B 0,C 180,E1 -27454.787,E2 -27454.787} C_VEL
LIN {X 0,Y 84.92,Z 305.435,A -85,B 0,C 180,E1 -27464.376,E2 -27464.376} C_VEL
LIN {X 0,Y 87.835,Z 304.904,A -85,B 0,C 180,E1 -27473.582,E2 -27473.582} C_VEL
LIN {X 0,Y 90.206,Z 304.062,A -85,B 0,C 180,E1 -27477.87,E2 -27477.87} C_VEL
LIN {X 0,Y 96.364,Z 301.141,A -85,B 0,C 180,E1 -27485.694,E2 -27485.694} C_VEL
LIN {X 0,Y 101.939,Z 297.851,A -85,B 0,C 180,E1 -27490.914,E2 -27490.914} C_VEL
LIN {X 0,Y 108.342,Z 293.522,A -85,B 0,C 180,E1 -27495.525,E2 -27495.525} C_VEL
LIN {X 0,Y 116.709,Z 287.025,A -85,B 0,C 180,E1 -27500.155,E2 -27500.155} C_VEL
LIN {X 0,Y 124.495,Z 279.947,A -85,B 0,C 180,E1 -27503.557,E2 -27503.557} C_VEL
LIN {X 0,Y 132.671,Z 271.141,A -85,B 0,C 180,E1 -27506.546,E2 -27506.546} C_VEL
LIN {X 0,Y 140.5,Z 261.168,A -85,B 0,C 180,E1 -27508.939,E2 -27508.939} C_VEL
LIN {X 0,Y 147.138,Z 251.012,A -85,B 0,C 180,E1 -27510.658,E2 -27510.658} C_VEL
LIN {X 0,Y 153.191,Z 239.76,A -85,B 0,C 180,E1 -27512.024,E2 -27512.024} C_VEL
LIN {X 0,Y 158.423,Z 227.406,A -85,B 0,C 180,E1 -27513.129,E2 -27513.129} C_VEL
LIN {X 0,Y 162.445,Z 214.489,A -85,B 0,C 180,E1 -27513.932,E2 -27513.932} C_VEL
LIN {X 0,Y 165.206,Z 201.301,A -85,B 0,C 180,E1 -27514.487,E2 -27514.487} C_VEL
LIN {X 0,Y 165.75,Z 197.149,A -85,B 0,C 180,E1 -27514.652,E2 -27514.652} C_VEL
LIN {X 0,Y 163.947,Z 190.571,A -85,B 0,C 180,E1 -27517.306,E2 -27517.306} C_VEL
LIN {X 0,Y 162.84,Z 187.037,A -85,B 0,C 180,E1 -27519.057,E2 -27519.057} C_VEL
LIN {X 0,Y 161.696,Z 184.594,A -85,B 0,C 180,E1 -27520.912,E2 -27520.912} C_VEL
LIN {X 0,Y 160.491,Z 183.291,A -85,B 0,C 180,E1 -27522.933,E2 -27522.933} C_VEL
LIN {X 0,Y 157.526,Z 181.758,A -85,B 0,C 180,E1 -27530.156,E2 -27530.156} C_VEL
LIN {X 0,Y 156.931,Z 181.139,A -85,B 0,C 180,E1 -27534.861,E2 -27534.861} C_VEL
LIN {X 0,Y 157.306,Z 181.207,A -85,B 0,C 180,E1 -27539.36,E2 -27539.36} C_VEL
LIN {X 0,Y 157.677,Z 181.949,A -85,B 0,C 180,E1 -27541.277,E2 -27541.277} C_VEL
LIN {X 0,Y 159.077,Z 185.525,A -85,B 0,C 180,E1 -27545.864,E2 -27545.864} C_VEL
LIN {X 0,Y 160.716,Z 189.352,A -85,B 0,C 180,E1 -27549.359,E2 -27549.359} C_VEL
LIN {X 0,Y 162.762,Z 194.441,A -85,B 0,C 180,E1 -27552.933,E2 -27552.933} C_VEL
LIN {X 0,Y 163.238,Z 195.826,A -85,B 0,C 180,E1 -27553.76,E2 -27553.76} C_VEL
LIN {X 0,Y 160.584,Z 208.664,A -85,B 0,C 180,E1 -27554.426,E2 -27554.426} C_VEL
LIN {X 0,Y 156.98,Z 220.557,A -85,B 0,C 180,E1 -27555.305,E2 -27555.305} C_VEL
LIN {X 0,Y 152.079,Z 232.458,A -85,B 0,C 180,E1 -27556.48,E2 -27556.48} C_VEL
LIN {X 0,Y 145.966,Z 244.058,A -85,B 0,C 180,E1 -27558.024,E2 -27558.024} C_VEL
LIN {X 0,Y 139.909,Z 253.372,A -85,B 0,C 180,E1 -27559.633,E2 -27559.633} C_VEL
LIN {X 0,Y 132.727,Z 262.766,A -85,B 0,C 180,E1 -27561.934,E2 -27561.934} C_VEL
LIN {X 0,Y 124.069,Z 271.997,A -85,B 0,C 180,E1 -27564.996,E2 -27564.996} C_VEL
LIN {X 0,Y 115.925,Z 279.292,A -85,B 0,C 180,E1 -27568.469,E2 -27568.469} C_VEL
LIN {X 0,Y 108.244,Z 285.065,A -85,B 0,C 180,E1 -27572.429,E2 -27572.429} C_VEL
LIN {X 0,Y 101.091,Z 289.563,A -85,B 0,C 180,E1 -27576.918,E2 -27576.918} C_VEL
LIN {X 0,Y 94.641,Z 292.941,A -85,B 0,C 180,E1 -27582.047,E2 -27582.047} C_VEL
LIN {X 0,Y 90.776,Z 294.597,A -85,B 0,C 180,E1 -27585.83,E2 -27585.83} C_VEL
LIN {X 0,Y 87.343,Z 295.837,A -85,B 0,C 180,E1 -27589.931,E2 -27589.931} C_VEL
LIN {X 0,Y 84.335,Z 296.674,A -85,B 0,C 180,E1 -27594.314,E2 -27594.314} C_VEL
LIN {X 0,Y 81.613,Z 297.072,A -85,B 0,C 180,E1 -27599.444,E2 -27599.444} C_VEL
LIN {X 0,Y 78.28,Z 296.653,A -85,B 0,C 180,E1 -27608.954,E2 -27608.954} C_VEL
LIN {X 0,Y 77.349,Z 295.858,A -85,B 0,C 180,E1 -27614.182,E2 -27614.182} C_VEL
LIN {X 0,Y 77.018,Z 294.612,A -85,B 0,C 180,E1 -27619.485,E2 -27619.485} C_VEL
LIN {X 0,Y 77.471,Z 292.436,A -85,B 0,C 180,E1 -27626.272,E2 -27626.272} C_VEL
LIN {X 0,Y 78.877,Z 288.39,A -85,B 0,C 180,E1 -27635.112,E2 -27635.112} C_VEL
LIN {X 0,Y 81.386,Z 283.688,A -85,B 0,C 180,E1 -27642.468,E2 -27642.468} C_VEL
LIN {X 0,Y 85.56,Z 276.642,A -85,B 0,C 180,E1 -27650.433,E2 -27650.433} C_VEL
LIN {X 0,Y 90.35,Z 268.986,A -85,B 0,C 180,E1 -27656.569,E2 -27656.569} C_VEL
LIN {X 0,Y 95.835,Z 259.39,A -85,B 0,C 180,E1 -27662.119,E2 -27662.119} C_VEL
LIN {X 0,Y 101.152,Z 249.456,A -85,B 0,C 180,E1 -27666.199,E2 -27666.199} C_VEL
LIN {X 0,Y 106.287,Z 238.235,A -85,B 0,C 180,E1 -27669.527,E2 -27669.527} C_VEL
LIN {X 0,Y 110.405,Z 227.271,A -85,B 0,C 180,E1 -27671.944,E2 -27671.944} C_VEL
LIN {X 0,Y 114.133,Z 214.437,A -85,B 0,C 180,E1 -27674.046,E2 -27674.046} C_VEL
LIN {X 0,Y 116.827,Z 200.939,A -85,B 0,C 180,E1 -27675.572,E2 -27675.572} C_VEL
LIN {X 0,Y 118.453,Z 187.968,A -85,B 0,C 180,E1 -27676.472,E2 -27676.472} C_VEL
LIN {X 0,Y 120.812,Z 159.376,A -85,B 0,C 180,E1 -27677.796,E2 -27677.796} C_VEL
LIN {X 0,Y 117.186,Z 151.298,A -85,B 0,C 180,E1 -27681.143,E2 -27681.143} C_VEL
LIN {X 0,Y 113.308,Z 144.144,A -85,B 0,C 180,E1 -27685.177,E2 -27685.177} C_VEL
LIN {X 0,Y 110.228,Z 138.926,A -85,B 0,C 180,E1 -27688.942,E2 -27688.942} C_VEL
LIN {X 0,Y 107.858,Z 135.191,A -85,B 0,C 180,E1 -27692.359,E2 -27692.359} C_VEL
LIN {X 0,Y 105.549,Z 131.512,A -85,B 0,C 180,E1 -27696.453,E2 -27696.453} C_VEL
LIN {X 0,Y 103.24,Z 128.39,A -85,B 0,C 180,E1 -27701.862,E2 -27701.862} C_VEL
LIN {X 0,Y 102.629,Z 126.718,A -85,B 0,C 180,E1 -27704.103,E2 -27704.103} C_VEL
LIN {X 0,Y 101.077,Z 125.501,A -85,B 0,C 180,E1 -27714.014,E2 -27714.014} C_VEL
LIN {X 0,Y 101.62,Z 125.688,A -85,B 0,C 180,E1 -27720.743,E2 -27720.743} C_VEL
LIN {X 0,Y 102.913,Z 126.879,A -85,B 0,C 180,E1 -27726.034,E2 -27726.034} C_VEL
LIN {X 0,Y 104.701,Z 130.477,A -85,B 0,C 180,E1 -27731.066,E2 -27731.066} C_VEL
LIN {X 0,Y 105.901,Z 131.823,A -85,B 0,C 180,E1 -27733.432,E2 -27733.432} C_VEL
LIN {X 0,Y 108.153,Z 135.401,A -85,B 0,C 180,E1 -27737.308,E2 -27737.308} C_VEL
LIN {X 0,Y 111.514,Z 140.95,A -85,B 0,C 180,E1 -27741.945,E2 -27741.945} C_VEL
LIN {X 0,Y 115.113,Z 147.352,A -85,B 0,C 180,E1 -27746.029,E2 -27746.029} C_VEL
LIN {X 0,Y 116.586,Z 151.095,A -85,B 0,C 180,E1 -27747.631,E2 -27747.631} C_VEL
LIN {X 0,Y 119.451,Z 160.135,A -85,B 0,C 180,E1 -27750.639,E2 -27750.639} C_VEL
LIN {X 0,Y 120.019,Z 162.83,A -85,B 0,C 180,E1 -27751.283,E2 -27751.283} C_VEL
LIN {X 0,Y 119.853,Z 172.446,A -85,B 0,C 180,E1 -27752.126,E2 -27752.126} C_VEL
LIN {X 0,Y 117.147,Z 202.202,A -85,B 0,C 180,E1 -27753.532,E2 -27753.532} C_VEL
LIN {X 0,Y 114.655,Z 216.084,A -85,B 0,C 180,E1 -27754.657,E2 -27754.657} C_VEL
LIN {X 0,Y 111.524,Z 228.056,A -85,B 0,C 180,E1 -27756.155,E2 -27756.155} C_VEL
LIN {X 0,Y 107.333,Z 239.927,A -85,B 0,C 180,E1 -27758.21,E2 -27758.21} C_VEL
LIN {X 0,Y 102.472,Z 251.375,A -85,B 0,C 180,E1 -27761.024,E2 -27761.024} C_VEL
LIN {X 0,Y 97.264,Z 261.665,A -85,B 0,C 180,E1 -27764.476,E2 -27764.476} C_VEL
LIN {X 0,Y 91.76,Z 271.778,A -85,B 0,C 180,E1 -27769.38,E2 -27769.38} C_VEL
LIN {X 0,Y 86.31,Z 280.631,A -85,B 0,C 180,E1 -27775.249,E2 -27775.249} C_VEL
LIN {X 0,Y 82.31,Z 287.737,A -85,B 0,C 180,E1 -27781.99,E2 -27781.99} C_VEL
LIN {X 0,Y 79.23,Z 293.387,A -85,B 0,C 180,E1 -27789.217,E2 -27789.217} C_VEL
LIN {X 0,Y 77.537,Z 297.827,A -85,B 0,C 180,E1 -27796.902,E2 -27796.902} C_VEL
LIN {X 0,Y 77.041,Z 301.158,A -85,B 0,C 180,E1 -27804.765,E2 -27804.765} C_VEL
LIN {X 0,Y 77.309,Z 302.802,A -85,B 0,C 180,E1 -27810,E2 -27810} C_VEL
LIN {X 0,Y 77.125,Z 303.968,A -85,B 0,C 180,E1 -27815.228,E2 -27815.228} C_VEL
LIN {X 0,Y 77.284,Z 304.712,A -85,B 0,C 180,E1 -27820.479,E2 -27820.479} C_VEL
LIN {X 0,Y 79.404,Z 304.984,A -85,B 0,C 180,E1 -27830.734,E2 -27830.734} C_VEL
LIN {X 0,Y 83.974,Z 303.759,A -85,B 0,C 180,E1 -27840.143,E2 -27840.143} C_VEL
LIN {X 0,Y 87.067,Z 302.531,A -85,B 0,C 180,E1 -27844.405,E2 -27844.405} C_VEL
LIN {X 0,Y 93.32,Z 299.52,A -85,B 0,C 180,E1 -27850.926,E2 -27850.926} C_VEL
LIN {X 0,Y 101.139,Z 294.949,A -85,B 0,C 180,E1 -27856.855,E2 -27856.855} C_VEL
LIN {X 0,Y 108.408,Z 289.935,A -85,B 0,C 180,E1 -27861.073,E2 -27861.073} C_VEL
LIN {X 0,Y 116.298,Z 283.672,A -85,B 0,C 180,E1 -27864.668,E2 -27864.668} C_VEL
LIN {X 0,Y 124.586,Z 275.885,A -85,B 0,C 180,E1 -27867.797,E2 -27867.797} C_VEL
LIN {X 0,Y 133.298,Z 266.173,A -85,B 0,C 180,E1 -27870.453,E2 -27870.453} C_VEL
LIN {X 0,Y 140.81,Z 256.155,A -85,B 0,C 180,E1 -27872.366,E2 -27872.366} C_VEL
LIN {X 0,Y 146.916,Z 246.262,A -85,B 0,C 180,E1 -27873.759,E2 -27873.759} C_VEL
LIN {X 0,Y 153.13,Z 233.766,A -85,B 0,C 180,E1 -27875.018,E2 -27875.018} C_VEL
LIN {X 0,Y 157.584,Z 222.16,A -85,B 0,C 180,E1 -27875.872,E2 -27875.872} C_VEL
LIN {X 0,Y 161.142,Z 209.499,A -85,B 0,C 180,E1 -27876.512,E2 -27876.512} C_VEL
LIN {X 0,Y 162.886,Z 200.232,A -85,B 0,C 180,E1 -27876.896,E2 -27876.896} C_VEL
LIN {X 0,Y 161.16,Z 193.191,A -85,B 0,C 180,E1 -27880.164,E2 -27880.164} C_VEL
LIN {X 0,Y 159.477,Z 187.362,A -85,B 0,C 180,E1 -27883.765,E2 -27883.765} C_VEL
LIN {X 0,Y 158.58,Z 184.702,A -85,B 0,C 180,E1 -27886.152,E2 -27886.152} C_VEL
LIN {X 0,Y 157.526,Z 181.758,A -85,B 0,C 180,E1 -27890.156,E2 -27890.156} C_VEL
LIN {X 0,Y 157.101,Z 181.667,A -85,B 0,C 180,E1 -27892.297,E2 -27892.297} C_VEL
LIN {X 0,Y 156.755,Z 182.763,A -85,B 0,C 180,E1 -27894.424,E2 -27894.424} C_VEL
LIN {X 0,Y 156.791,Z 189.41,A -85,B 0,C 180,E1 -27901.416,E2 -27901.416} C_VEL
LIN {X 0,Y 157.854,Z 192.378,A -85,B 0,C 180,E1 -27905.268,E2 -27905.268} C_VEL
LIN {X 0,Y 159.116,Z 195.971,A -85,B 0,C 180,E1 -27908.573,E2 -27908.573} C_VEL
LIN {X 0,Y 160.423,Z 199.902,A -85,B 0,C 180,E1 -27911.489,E2 -27911.489} C_VEL
LIN {X 0,Y 157.253,Z 212.948,A -85,B 0,C 180,E1 -27912.248,E2 -27912.248} C_VEL
LIN {X 0,Y 153.299,Z 224.436,A -85,B 0,C 180,E1 -27913.148,E2 -27913.148} C_VEL
LIN {X 0,Y 148.611,Z 234.898,A -85,B 0,C 180,E1 -27914.193,E2 -27914.193} C_VEL
LIN {X 0,Y 142.322,Z 246.079,A -85,B 0,C 180,E1 -27915.649,E2 -27915.649} C_VEL
LIN {X 0,Y 136.103,Z 255.09,A -85,B 0,C 180,E1 -27917.197,E2 -27917.197} C_VEL
LIN {X 0,Y 128.266,Z 264.666,A -85,B 0,C 180,E1 -27919.572,E2 -27919.572} C_VEL
LIN {X 0,Y 119.729,Z 273.243,A -85,B 0,C 180,E1 -27922.405,E2 -27922.405} C_VEL
LIN {X 0,Y 111.25,Z 280.344,A -85,B 0,C 180,E1 -27925.814,E2 -27925.814} C_VEL
LIN {X 0,Y 101.923,Z 286.77,A -85,B 0,C 180,E1 -27930.466,E2 -27930.466} C_VEL
LIN {X 0,Y 94.505,Z 290.959,A -85,B 0,C 180,E1 -27935.112,E2 -27935.112} C_VEL
LIN {X 0,Y 89.731,Z 293.25,A -85,B 0,C 180,E1 -27938.798,E2 -27938.798} C_VEL
LIN {X 0,Y 81.901,Z 296.125,A -85,B 0,C 180,E1 -27946.648,E2 -27946.648} C_VEL
LIN {X 0,Y 78.54,Z 296.995,A -85,B 0,C 180,E1 -27951.217,E2 -27951.217} C_VEL
LIN {X 0,Y 75.068,Z 297.468,A -85,B 0,C 180,E1 -27957.414,E2 -27957.414} C_VEL
LIN {X 0,Y 71.599,Z 297.089,A -85,B 0,C 180,E1 -27966.882,E2 -27966.882} C_VEL
LIN {X 0,Y 70.436,Z 296.332,A -85,B 0,C 180,E1 -27972.583,E2 -27972.583} C_VEL
LIN {X 0,Y 69.951,Z 295.138,A -85,B 0,C 180,E1 -27978.408,E2 -27978.408} C_VEL
LIN {X 0,Y 70.396,Z 292.73,A -85,B 0,C 180,E1 -27986.697,E2 -27986.697} C_VEL
LIN {X 0,Y 71.808,Z 289.038,A -85,B 0,C 180,E1 -27995.617,E2 -27995.617} C_VEL
LIN {X 0,Y 74.478,Z 284.407,A -85,B 0,C 180,E1 -28003.646,E2 -28003.646} C_VEL
LIN {X 0,Y 78.951,Z 277.44,A -85,B 0,C 180,E1 -28012.23,E2 -28012.23} C_VEL
LIN {X 0,Y 84.082,Z 269.887,A -85,B 0,C 180,E1 -28018.726,E2 -28018.726} C_VEL
LIN {X 0,Y 88.891,Z 262.191,A -85,B 0,C 180,E1 -28023.604,E2 -28023.604} C_VEL
LIN {X 0,Y 94.342,Z 252.776,A -85,B 0,C 180,E1 -28027.923,E2 -28027.923} C_VEL
LIN {X 0,Y 99.703,Z 242.304,A -85,B 0,C 180,E1 -28031.365,E2 -28031.365} C_VEL
LIN {X 0,Y 104.649,Z 230.677,A -85,B 0,C 180,E1 -28034.169,E2 -28034.169} C_VEL
LIN {X 0,Y 108.675,Z 218.425,A -85,B 0,C 180,E1 -28036.317,E2 -28036.317} C_VEL
LIN {X 0,Y 111.79,Z 205.222,A -85,B 0,C 180,E1 -28038,E2 -28038} C_VEL
LIN {X 0,Y 113.756,Z 192.722,A -85,B 0,C 180,E1 -28039.023,E2 -28039.023} C_VEL
LIN {X 0,Y 116.483,Z 162.12,A -85,B 0,C 180,E1 -28040.475,E2 -28040.475} C_VEL
LIN {X 0,Y 113.451,Z 155.228,A -85,B 0,C 180,E1 -28043.664,E2 -28043.664} C_VEL
LIN {X 0,Y 109.911,Z 148.279,A -85,B 0,C 180,E1 -28047.911,E2 -28047.911} C_VEL
LIN {X 0,Y 107.473,Z 144.113,A -85,B 0,C 180,E1 -28051.326,E2 -28051.326} C_VEL
LIN {X 0,Y 106.03,Z 141.593,A -85,B 0,C 180,E1 -28053.688,E2 -28053.688} C_VEL
LIN {X 0,Y 103.882,Z 138.029,A -85,B 0,C 180,E1 -28057.894,E2 -28057.894} C_VEL
LIN {X 0,Y 101.862,Z 134.817,A -85,B 0,C 180,E1 -28063.361,E2 -28063.361} C_VEL
LIN {X 0,Y 101.449,Z 133.618,A -85,B 0,C 180,E1 -28065.11,E2 -28065.11} C_VEL
LIN {X 0,Y 100.207,Z 132.553,A -85,B 0,C 180,E1 -28073.962,E2 -28073.962} C_VEL
LIN {X 0,Y 100.63,Z 132.611,A -85,B 0,C 180,E1 -28080,E2 -28080} C_VEL
LIN {X 0,Y 101.751,Z 133.829,A -85,B 0,C 180,E1 -28085.202,E2 -28085.202} C_VEL
LIN {X 0,Y 103.337,Z 137.211,A -85,B 0,C 180,E1 -28090.099,E2 -28090.099} C_VEL
LIN {X 0,Y 104.387,Z 138.633,A -85,B 0,C 180,E1 -28092.393,E2 -28092.393} C_VEL
LIN {X 0,Y 106.886,Z 142.917,A -85,B 0,C 180,E1 -28096.965,E2 -28096.965} C_VEL
LIN {X 0,Y 110.03,Z 148.425,A -85,B 0,C 180,E1 -28101.487,E2 -28101.487} C_VEL
LIN {X 0,Y 112.685,Z 153.817,A -85,B 0,C 180,E1 -28104.746,E2 -28104.746} C_VEL
LIN {X 0,Y 115.388,Z 162.766,A -85,B 0,C 180,E1 -28108.028,E2 -28108.028} C_VEL
LIN {X 0,Y 115.878,Z 164.955,A -85,B 0,C 180,E1 -28108.639,E2 -28108.639} C_VEL
LIN {X 0,Y 115.664,Z 173.013,A -85,B 0,C 180,E1 -28109.362,E2 -28109.362} C_VEL
LIN {X 0,Y 112.988,Z 201.165,A -85,B 0,C 180,E1 -28110.66,E2 -28110.66} C_VEL
LIN {X 0,Y 110.527,Z 214.569,A -85,B 0,C 180,E1 -28111.687,E2 -28111.687} C_VEL
LIN {X 0,Y 107.129,Z 227.335,A -85,B 0,C 180,E1 -28113.232,E2 -28113.232} C_VEL
LIN {X 0,Y 103.037,Z 238.476,A -85,B 0,C 180,E1 -28115.064,E2 -28115.064} C_VEL
LIN {X 0,Y 97.966,Z 250.138,A -85,B 0,C 180,E1 -28117.894,E2 -28117.894} C_VEL
LIN {X 0,Y 92.351,Z 260.577,A -85,B 0,C 180,E1 -28121.279,E2 -28121.279} C_VEL
LIN {X 0,Y 87.468,Z 269.172,A -85,B 0,C 180,E1 -28125.326,E2 -28125.326} C_VEL
LIN {X 0,Y 82.58,Z 276.736,A -85,B 0,C 180,E1 -28129.992,E2 -28129.992} C_VEL
LIN {X 0,Y 79.716,Z 281.108,A -85,B 0,C 180,E1 -28133.479,E2 -28133.479} C_VEL
LIN {X 0,Y 75.402,Z 288.038,A -85,B 0,C 180,E1 -28140.702,E2 -28140.702} C_VEL
LIN {X 0,Y 71.765,Z 294.374,A -85,B 0,C 180,E1 -28149.954,E2 -28149.954} C_VEL
LIN {X 0,Y 70.256,Z 298.497,A -85,B 0,C 180,E1 -28158.459,E2 -28158.459} C_VEL
LIN {X 0,Y 69.967,Z 300.626,A -85,B 0,C 180,E1 -28164.235,E2 -28164.235} C_VEL
LIN {X 0,Y 70.2,Z 302.296,A -85,B 0,C 180,E1 -28170,E2 -28170} C_VEL
LIN {X 0,Y 70.045,Z 303.49,A -85,B 0,C 180,E1 -28175.758,E2 -28175.758} C_VEL
LIN {X 0,Y 70.291,Z 304.275,A -85,B 0,C 180,E1 -28181.535,E2 -28181.535} C_VEL
LIN {X 0,Y 72.78,Z 304.611,A -85,B 0,C 180,E1 -28192.722,E2 -28192.722} C_VEL
LIN {X 0,Y 77.899,Z 303.442,A -85,B 0,C 180,E1 -28202.773,E2 -28202.773} C_VEL
LIN {X 0,Y 81.287,Z 302.264,A -85,B 0,C 180,E1 -28207.244,E2 -28207.244} C_VEL
LIN {X 0,Y 88.847,Z 298.919,A -85,B 0,C 180,E1 -28214.608,E2 -28214.608} C_VEL
LIN {X 0,Y 96.398,Z 294.798,A -85,B 0,C 180,E1 -28219.953,E2 -28219.953} C_VEL
LIN {X 0,Y 104.086,Z 289.849,A -85,B 0,C 180,E1 -28224.121,E2 -28224.121} C_VEL
LIN {X 0,Y 112.349,Z 283.655,A -85,B 0,C 180,E1 -28227.618,E2 -28227.618} C_VEL
LIN {X 0,Y 120.955,Z 275.984,A -85,B 0,C 180,E1 -28230.641,E2 -28230.641} C_VEL
LIN {X 0,Y 129.95,Z 266.375,A -85,B 0,C 180,E1 -28233.172,E2 -28233.172} C_VEL
LIN {X 0,Y 137.672,Z 256.484,A -85,B 0,C 180,E1 -28234.975,E2 -28234.975} C_VEL
LIN {X 0,Y 143.926,Z 246.786,A -85,B 0,C 180,E1 -28236.288,E2 -28236.288} C_VEL
LIN {X 0,Y 149.494,Z 236.316,A -85,B 0,C 180,E1 -28237.311,E2 -28237.311} C_VEL
LIN {X 0,Y 154.514,Z 224.204,A -85,B 0,C 180,E1 -28238.194,E2 -28238.194} C_VEL
LIN {X 0,Y 158.479,Z 211.298,A -85,B 0,C 180,E1 -28238.842,E2 -28238.842} C_VEL
LIN {X 0,Y 160.137,Z 203.564,A -85,B 0,C 180,E1 -28239.194,E2 -28239.194} C_VEL
LIN {X 0,Y 159.015,Z 197.654,A -85,B 0,C 180,E1 -28242.227,E2 -28242.227} C_VEL
LIN {X 0,Y 157.959,Z 193.275,A -85,B 0,C 180,E1 -28245.177,E2 -28245.177} C_VEL
LIN {X 0,Y 157.353,Z 191.278,A -85,B 0,C 180,E1 -28247.096,E2 -28247.096} C_VEL
LIN {X 0,Y 156.503,Z 188.639,A -85,B 0,C 180,E1 -28250.867,E2 -28250.867} C_VEL
LIN {X 0,Y 156.174,Z 188.031,A -85,B 0,C 180,E1 -28257.42,E2 -28257.42} C_VEL
LIN {X 0,Y 156.659,Z 188.757,A -85,B 0,C 180,E1 -28260.642,E2 -28260.642} C_VEL
LIN {X 0,Y 156.791,Z 189.41,A -85,B 0,C 180,E1 -28261.416,E2 -28261.416} C_VEL
LIN {X 0,Y 156.99,Z 191.113,A -85,B 0,C 180,E1 -28262.717,E2 -28262.717} C_VEL
LIN {X 0,Y 157.036,Z 195.524,A -85,B 0,C 180,E1 -28264.553,E2 -28264.553} C_VEL
LIN {X 0,Y 156.988,Z 200.186,A -85,B 0,C 180,E1 -28266.358,E2 -28266.358} C_VEL
LIN {X 0,Y 157.182,Z 202.267,A -85,B 0,C 180,E1 -28267.615,E2 -28267.615} C_VEL
LIN {X 0,Y 157.692,Z 204.323,A -85,B 0,C 180,E1 -28269.248,E2 -28269.248} C_VEL
LIN {X 0,Y 154.344,Z 216.42,A -85,B 0,C 180,E1 -28269.96,E2 -28269.96} C_VEL
LIN {X 0,Y 149.839,Z 228.124,A -85,B 0,C 180,E1 -28270.881,E2 -28270.881} C_VEL
LIN {X 0,Y 143.767,Z 240.187,A -85,B 0,C 180,E1 -28272.123,E2 -28272.123} C_VEL
LIN {X 0,Y 137.324,Z 250.374,A -85,B 0,C 180,E1 -28273.494,E2 -28273.494} C_VEL
LIN {X 0,Y 129.766,Z 260.205,A -85,B 0,C 180,E1 -28275.39,E2 -28275.39} C_VEL
LIN {X 0,Y 121.737,Z 268.874,A -85,B 0,C 180,E1 -28277.718,E2 -28277.718} C_VEL
LIN {X 0,Y 112.679,Z 276.954,A -85,B 0,C 180,E1 -28280.679,E2 -28280.679} C_VEL
LIN {X 0,Y 105.13,Z 282.58,A -85,B 0,C 180,E1 -28283.647,E2 -28283.647} C_VEL
LIN {X 0,Y 95.728,Z 288.421,A -85,B 0,C 180,E1 -28288.238,E2 -28288.238} C_VEL
LIN {X 0,Y 88.012,Z 292.297,A -85,B 0,C 180,E1 -28293.023,E2 -28293.023} C_VEL
LIN {X 0,Y 80.992,Z 295.107,A -85,B 0,C 180,E1 -28298.651,E2 -28298.651} C_VEL
LIN {X 0,Y 76.77,Z 296.412,A -85,B 0,C 180,E1 -28302.915,E2 -28302.915} C_VEL
LIN {X 0,Y 73.028,Z 297.312,A -85,B 0,C 180,E1 -28307.65,E2 -28307.65} C_VEL
LIN {X 0,Y 68.676,Z 297.861,A -85,B 0,C 180,E1 -28314.953,E2 -28314.953} C_VEL
LIN {X 0,Y 65.006,Z 297.526,A -85,B 0,C 180,E1 -28324.377,E2 -28324.377} C_VEL
LIN {X 0,Y 63.581,Z 296.798,A -85,B 0,C 180,E1 -28330.634,E2 -28330.634} C_VEL
LIN {X 0,Y 62.9,Z 295.664,A -85,B 0,C 180,E1 -28337.088,E2 -28337.088} C_VEL
LIN {X 0,Y 63.329,Z 293.04,A -85,B 0,C 180,E1 -28347.154,E2 -28347.154} C_VEL
LIN {X 0,Y 64.748,Z 289.671,A -85,B 0,C 180,E1 -28356.232,E2 -28356.232} C_VEL
LIN {X 0,Y 67.607,Z 285.116,A -85,B 0,C 180,E1 -28365.064,E2 -28365.064} C_VEL
LIN {X 0,Y 72.44,Z 278.237,A -85,B 0,C 180,E1 -28374.352,E2 -28374.352} C_VEL
LIN {X 0,Y 77.929,Z 270.774,A -85,B 0,C 180,E1 -28381.237,E2 -28381.237} C_VEL
LIN {X 0,Y 83.103,Z 263.176,A -85,B 0,C 180,E1 -28386.299,E2 -28386.299} C_VEL
LIN {X 0,Y 88.853,Z 253.951,A -85,B 0,C 180,E1 -28390.735,E2 -28390.735} C_VEL
LIN {X 0,Y 94.5,Z 243.645,A -85,B 0,C 180,E1 -28394.205,E2 -28394.205} C_VEL
LIN {X 0,Y 99.717,Z 232.227,A -85,B 0,C 180,E1 -28396.99,E2 -28396.99} C_VEL
LIN {X 0,Y 103.958,Z 220.373,A -85,B 0,C 180,E1 -28399.142,E2 -28399.142} C_VEL
LIN {X 0,Y 107.354,Z 207.274,A -85,B 0,C 180,E1 -28400.838,E2 -28400.838} C_VEL
LIN {X 0,Y 109.648,Z 194.015,A -85,B 0,C 180,E1 -28401.973,E2 -28401.973} C_VEL
LIN {X 0,Y 112.435,Z 165.6,A -85,B 0,C 180,E1 -28403.259,E2 -28403.259} C_VEL
LIN {X 0,Y 112.215,Z 164.39,A -85,B 0,C 180,E1 -28403.595,E2 -28403.595} C_VEL
LIN {X 0,Y 108.995,Z 157.103,A -85,B 0,C 180,E1 -28407.594,E2 -28407.594} C_VEL
LIN {X 0,Y 106.084,Z 151.345,A -85,B 0,C 180,E1 -28411.856,E2 -28411.856} C_VEL
LIN {X 0,Y 103.98,Z 147.591,A -85,B 0,C 180,E1 -28415.59,E2 -28415.59} C_VEL
LIN {X 0,Y 102.268,Z 144.491,A -85,B 0,C 180,E1 -28419.426,E2 -28419.426} C_VEL
LIN {X 0,Y 100.507,Z 141.078,A -85,B 0,C 180,E1 -28425.135,E2 -28425.135} C_VEL
LIN {X 0,Y 100.351,Z 140.553,A -85,B 0,C 180,E1 -28425.934,E2 -28425.934} C_VEL
LIN {X 0,Y 99.376,Z 139.439,A -85,B 0,C 180,E1 -28435.945,E2 -28435.945} C_VEL
LIN {X 0,Y 99.991,Z 140.001,A -85,B 0,C 180,E1 -28441.511,E2 -28441.511} C_VEL
LIN {X 0,Y 100.586,Z 140.765,A -85,B 0,C 180,E1 -28444.258,E2 -28444.258} C_VEL
LIN {X 0,Y 102.315,Z 144.372,A -85,B 0,C 180,E1 -28449.889,E2 -28449.889} C_VEL
LIN {X 0,Y 103.381,Z 146.381,A -85,B 0,C 180,E1 -28452.391,E2 -28452.391} C_VEL
LIN {X 0,Y 105.059,Z 149.399,A -85,B 0,C 180,E1 -28455.645,E2 -28455.645} C_VEL
LIN {X 0,Y 107.743,Z 154.435,A -85,B 0,C 180,E1 -28459.903,E2 -28459.903} C_VEL
LIN {X 0,Y 109.774,Z 159.026,A -85,B 0,C 180,E1 -28462.715,E2 -28462.715} C_VEL
LIN {X 0,Y 111.961,Z 167.146,A -85,B 0,C 180,E1 -28465.778,E2 -28465.778} C_VEL
LIN {X 0,Y 111.73,Z 173.851,A -85,B 0,C 180,E1 -28466.403,E2 -28466.403} C_VEL
LIN {X 0,Y 108.866,Z 201.893,A -85,B 0,C 180,E1 -28467.688,E2 -28467.688} C_VEL
LIN {X 0,Y 106.123,Z 215.711,A -85,B 0,C 180,E1 -28468.758,E2 -28468.758} C_VEL
LIN {X 0,Y 102.345,Z 228.653,A -85,B 0,C 180,E1 -28470.381,E2 -28470.381} C_VEL
LIN {X 0,Y 97.764,Z 240.241,A -85,B 0,C 180,E1 -28472.362,E2 -28472.362} C_VEL
LIN {X 0,Y 92.406,Z 251.491,A -85,B 0,C 180,E1 -28475.153,E2 -28475.153} C_VEL
LIN {X 0,Y 86.605,Z 261.569,A -85,B 0,C 180,E1 -28478.64,E2 -28478.64} C_VEL
LIN {X 0,Y 80.322,Z 271.568,A -85,B 0,C 180,E1 -28483.791,E2 -28483.791} C_VEL
LIN {X 0,Y 74.007,Z 280.298,A -85,B 0,C 180,E1 -28490.132,E2 -28490.132} C_VEL
LIN {X 0,Y 69.24,Z 287.314,A -85,B 0,C 180,E1 -28497.799,E2 -28497.799} C_VEL
LIN {X 0,Y 65.092,Z 293.718,A -85,B 0,C 180,E1 -28507.796,E2 -28507.796} C_VEL
LIN {X 0,Y 63.275,Z 297.904,A -85,B 0,C 180,E1 -28517.164,E2 -28517.164} C_VEL
LIN {X 0,Y 62.89,Z 300.092,A -85,B 0,C 180,E1 -28523.583,E2 -28523.583} C_VEL
LIN {X 0,Y 63.102,Z 301.792,A -85,B 0,C 180,E1 -28529.999,E2 -28529.999} C_VEL
LIN {X 0,Y 62.97,Z 303.011,A -85,B 0,C 180,E1 -28536.408,E2 -28536.408} C_VEL
LIN {X 0,Y 63.339,Z 303.826,A -85,B 0,C 180,E1 -28542.821,E2 -28542.821} C_VEL
LIN {X 0,Y 64.426,Z 304.236,A -85,B 0,C 180,E1 -28549.102,E2 -28549.102} C_VEL
LIN {X 0,Y 68.775,Z 303.864,A -85,B 0,C 180,E1 -28560.726,E2 -28560.726} C_VEL
LIN {X 0,Y 75.739,Z 301.992,A -85,B 0,C 180,E1 -28570.507,E2 -28570.507} C_VEL
LIN {X 0,Y 83.362,Z 298.972,A -85,B 0,C 180,E1 -28577.587,E2 -28577.587} C_VEL
LIN {X 0,Y 91.977,Z 294.647,A -85,B 0,C 180,E1 -28583.351,E2 -28583.351} C_VEL
LIN {X 0,Y 100.089,Z 289.763,A -85,B 0,C 180,E1 -28587.417,E2 -28587.417} C_VEL
LIN {X 0,Y 108.721,Z 283.644,A -85,B 0,C 180,E1 -28590.771,E2 -28590.771} C_VEL
LIN {X 0,Y 117.642,Z 276.068,A -85,B 0,C 180,E1 -28593.651,E2 -28593.651} C_VEL
LIN {X 0,Y 125.359,Z 268.353,A -85,B 0,C 180,E1 -28595.647,E2 -28595.647} C_VEL
LIN {X 0,Y 132.434,Z 260.014,A -85,B 0,C 180,E1 -28597.229,E2 -28597.229} C_VEL
LIN {X 0,Y 139.6,Z 249.871,A -85,B 0,C 180,E1 -28598.648,E2 -28598.648} C_VEL
LIN {X 0,Y 146.089,Z 238.63,A -85,B 0,C 180,E1 -28599.736,E2 -28599.736} C_VEL
LIN {X 0,Y 151.662,Z 226.344,A -85,B 0,C 180,E1 -28600.6,E2 -28600.6} C_VEL
LIN {X 0,Y 155.875,Z 213.716,A -85,B 0,C 180,E1 -28601.234,E2 -28601.234} C_VEL
LIN {X 0,Y 157.484,Z 207.433,A -85,B 0,C 180,E1 -28601.447,E2 -28601.447} C_VEL
LIN {X 0,Y 157.132,Z 203.76,A -85,B 0,C 180,E1 -28603.349,E2 -28603.349} C_VEL
LIN {X 0,Y 156.443,Z 199.64,A -85,B 0,C 180,E1 -28606.192,E2 -28606.192} C_VEL
LIN {X 0,Y 156.047,Z 197.884,A -85,B 0,C 180,E1 -28607.977,E2 -28607.977} C_VEL
LIN {X 0,Y 155.477,Z 195.613,A -85,B 0,C 180,E1 -28611.213,E2 -28611.213} C_VEL
LIN {X 0,Y 155.209,Z 195.041,A -85,B 0,C 180,E1 -28617.404,E2 -28617.404} C_VEL
LIN {X 0,Y 155.556,Z 195.693,A -85,B 0,C 180,E1 -28620.161,E2 -28620.161} C_VEL
LIN {X 0,Y 156.378,Z 199.156,A -85,B 0,C 180,E1 -28624.672,E2 -28624.672} C_VEL
LIN {X 0,Y 157.162,Z 202.188,A -85,B 0,C 180,E1 -28627.548,E2 -28627.548} C_VEL
LIN {X 0,Y 157.182,Z 202.267,A -85,B 0,C 180,E1 -28627.615,E2 -28627.615} C_VEL
LIN {X 0,Y 157.151,Z 203.888,A -85,B 0,C 180,E1 -28628.228,E2 -28628.228} C_VEL
LIN {X 0,Y 156.737,Z 206.172,A -85,B 0,C 180,E1 -28628.515,E2 -28628.515} C_VEL
LIN {X 0,Y 155.578,Z 210.072,A -85,B 0,C 180,E1 -28628.492,E2 -28628.492} C_VEL
LIN {X 0,Y 152.313,Z 218.323,A -85,B 0,C 180,E1 -28627.768,E2 -28627.768} C_VEL
LIN {X 0,Y 150.573,Z 222.511,A -85,B 0,C 180,E1 -28627.777,E2 -28627.777} C_VEL
LIN {X 0,Y 145.191,Z 234.422,A -85,B 0,C 180,E1 -28628.754,E2 -28628.754} C_VEL
LIN {X 0,Y 138.297,Z 246.316,A -85,B 0,C 180,E1 -28630.065,E2 -28630.065} C_VEL
LIN {X 0,Y 130.914,Z 256.427,A -85,B 0,C 180,E1 -28631.554,E2 -28631.554} C_VEL
LIN {X 0,Y 122.902,Z 265.553,A -85,B 0,C 180,E1 -28633.56,E2 -28633.56} C_VEL
LIN {X 0,Y 113.424,Z 274.399,A -85,B 0,C 180,E1 -28636.174,E2 -28636.174} C_VEL
LIN {X 0,Y 104.236,Z 281.401,A -85,B 0,C 180,E1 -28639.277,E2 -28639.277} C_VEL
LIN {X 0,Y 95.372,Z 286.959,A -85,B 0,C 180,E1 -28642.908,E2 -28642.908} C_VEL
LIN {X 0,Y 86.96,Z 291.283,A -85,B 0,C 180,E1 -28647.251,E2 -28647.251} C_VEL
LIN {X 0,Y 79.98,Z 294.2,A -85,B 0,C 180,E1 -28651.818,E2 -28651.818} C_VEL
LIN {X 0,Y 72.013,Z 296.702,A -85,B 0,C 180,E1 -28658.672,E2 -28658.672} C_VEL
LIN {X 0,Y 64.167,Z 298.163,A -85,B 0,C 180,E1 -28668.917,E2 -28668.917} C_VEL
LIN {X 0,Y 61.057,Z 298.271,A -85,B 0,C 180,E1 -28674.864,E2 -28674.864} C_VEL
LIN {X 0,Y 56.816,Z 297.265,A -85,B 0,C 180,E1 -28688.217,E2 -28688.217} C_VEL
LIN {X 0,Y 55.91,Z 296.173,A -85,B 0,C 180,E1 -28695.44,E2 -28695.44} C_VEL
LIN {X 0,Y 56.264,Z 293.319,A -85,B 0,C 180,E1 -28707.82,E2 -28707.82} C_VEL
LIN {X 0,Y 57.699,Z 290.286,A -85,B 0,C 180,E1 -28716.997,E2 -28716.997} C_VEL
LIN {X 0,Y 60.785,Z 285.804,A -85,B 0,C 180,E1 -28726.802,E2 -28726.802} C_VEL
LIN {X 0,Y 66.052,Z 279.033,A -85,B 0,C 180,E1 -28736.886,E2 -28736.886} C_VEL
LIN {X 0,Y 71.958,Z 271.66,A -85,B 0,C 180,E1 -28744.167,E2 -28744.167} C_VEL
LIN {X 0,Y 78.701,Z 262.51,A -85,B 0,C 180,E1 -28750.349,E2 -28750.349} C_VEL
LIN {X 0,Y 84.919,Z 252.987,A -85,B 0,C 180,E1 -28754.707,E2 -28754.707} C_VEL
LIN {X 0,Y 90.924,Z 242.401,A -85,B 0,C 180,E1 -28758.072,E2 -28758.072} C_VEL
LIN {X 0,Y 95.731,Z 232.201,A -85,B 0,C 180,E1 -28760.431,E2 -28760.431} C_VEL
LIN {X 0,Y 100.186,Z 220.181,A -85,B 0,C 180,E1 -28762.521,E2 -28762.521} C_VEL
LIN {X 0,Y 103.755,Z 206.868,A -85,B 0,C 180,E1 -28764.168,E2 -28764.168} C_VEL
LIN {X 0,Y 106.057,Z 193.918,A -85,B 0,C 180,E1 -28765.221,E2 -28765.221} C_VEL
LIN {X 0,Y 108.662,Z 167.981,A -85,B 0,C 180,E1 -28766.398,E2 -28766.398} C_VEL
LIN {X 0,Y 106.032,Z 161.715,A -85,B 0,C 180,E1 -28770.184,E2 -28770.184} C_VEL
LIN {X 0,Y 103.702,Z 156.771,A -85,B 0,C 180,E1 -28774.157,E2 -28774.157} C_VEL
LIN {X 0,Y 102.198,Z 153.811,A -85,B 0,C 180,E1 -28777.244,E2 -28777.244} C_VEL
LIN {X 0,Y 100.852,Z 151.119,A -85,B 0,C 180,E1 -28780.67,E2 -28780.67} C_VEL
LIN {X 0,Y 99.286,Z 147.504,A -85,B 0,C 180,E1 -28786.718,E2 -28786.718} C_VEL
LIN {X 0,Y 98.503,Z 146.497,A -85,B 0,C 180,E1 -28795.909,E2 -28795.909} C_VEL
LIN {X 0,Y 99.256,Z 147.257,A -85,B 0,C 180,E1 -28802.283,E2 -28802.283} C_VEL
LIN {X 0,Y 99.545,Z 148.019,A -85,B 0,C 180,E1 -28803.796,E2 -28803.796} C_VEL
LIN {X 0,Y 101.388,Z 151.957,A -85,B 0,C 180,E1 -28809.98,E2 -28809.98} C_VEL
LIN {X 0,Y 103.268,Z 155.811,A -85,B 0,C 180,E1 -28814.233,E2 -28814.233} C_VEL
LIN {X 0,Y 105.558,Z 160.586,A -85,B 0,C 180,E1 -28818.296,E2 -28818.296} C_VEL
LIN {X 0,Y 106.93,Z 163.872,A -85,B 0,C 180,E1 -28820.437,E2 -28820.437} C_VEL
LIN {X 0,Y 108.361,Z 169.812,A -85,B 0,C 180,E1 -28822.807,E2 -28822.807} C_VEL
LIN {X 0,Y 108.142,Z 174.452,A -85,B 0,C 180,E1 -28823.232,E2 -28823.232} C_VEL
LIN {X 0,Y 105.252,Z 201.35,A -85,B 0,C 180,E1 -28824.407,E2 -28824.407} C_VEL
LIN {X 0,Y 102.576,Z 214.511,A -85,B 0,C 180,E1 -28825.369,E2 -28825.369} C_VEL
LIN {X 0,Y 98.911,Z 226.935,A -85,B 0,C 180,E1 -28826.795,E2 -28826.795} C_VEL
LIN {X 0,Y 94.102,Z 238.788,A -85,B 0,C 180,E1 -28828.651,E2 -28828.651} C_VEL
LIN {X 0,Y 88.515,Z 250.256,A -85,B 0,C 180,E1 -28831.4,E2 -28831.4} C_VEL
LIN {X 0,Y 82.284,Z 260.518,A -85,B 0,C 180,E1 -28834.705,E2 -28834.705} C_VEL
LIN {X 0,Y 76.726,Z 268.985,A -85,B 0,C 180,E1 -28838.867,E2 -28838.867} C_VEL
LIN {X 0,Y 70.901,Z 276.667,A -85,B 0,C 180,E1 -28843.938,E2 -28843.938} C_VEL
LIN {X 0,Y 66.795,Z 282.02,A -85,B 0,C 180,E1 -28848.881,E2 -28848.881} C_VEL
LIN {X 0,Y 62.498,Z 287.614,A -85,B 0,C 180,E1 -28855.787,E2 -28855.787} C_VEL
LIN {X 0,Y 58.541,Z 293.063,A -85,B 0,C 180,E1 -28865.153,E2 -28865.153} C_VEL
LIN {X 0,Y 56.326,Z 297.31,A -85,B 0,C 180,E1 -28875.549,E2 -28875.549} C_VEL
LIN {X 0,Y 55.816,Z 299.551,A -85,B 0,C 180,E1 -28882.766,E2 -28882.766} C_VEL
LIN {X 0,Y 55.987,Z 301.286,A -85,B 0,C 180,E1 -28889.999,E2 -28889.999} C_VEL
LIN {X 0,Y 55.901,Z 302.532,A -85,B 0,C 180,E1 -28897.222,E2 -28897.222} C_VEL
LIN {X 0,Y 57.745,Z 303.829,A -85,B 0,C 180,E1 -28911.415,E2 -28911.415} C_VEL
LIN {X 0,Y 62.764,Z 303.518,A -85,B 0,C 180,E1 -28924.047,E2 -28924.047} C_VEL
LIN {X 0,Y 70.475,Z 301.706,A -85,B 0,C 180,E1 -28934.271,E2 -28934.271} C_VEL
LIN {X 0,Y 78.058,Z 299.039,A -85,B 0,C 180,E1 -28940.93,E2 -28940.93} C_VEL
LIN {X 0,Y 87.919,Z 294.505,A -85,B 0,C 180,E1 -28947.07,E2 -28947.07} C_VEL
LIN {X 0,Y 96.455,Z 289.689,A -85,B 0,C 180,E1 -28950.969,E2 -28950.969} C_VEL
LIN {X 0,Y 106.947,Z 282.521,A -85,B 0,C 180,E1 -28954.632,E2 -28954.632} C_VEL
LIN {X 0,Y 116.273,Z 274.744,A -85,B 0,C 180,E1 -28957.187,E2 -28957.187} C_VEL
LIN {X 0,Y 125.799,Z 265.045,A -85,B 0,C 180,E1 -28959.354,E2 -28959.354} C_VEL
LIN {X 0,Y 133.933,Z 255.041,A -85,B 0,C 180,E1 -28960.828,E2 -28960.828} C_VEL
LIN {X 0,Y 140.476,Z 245.171,A -85,B 0,C 180,E1 -28961.91,E2 -28961.91} C_VEL
LIN {X 0,Y 147.106,Z 232.695,A -85,B 0,C 180,E1 -28962.844,E2 -28962.844} C_VEL
LIN {X 0,Y 152.287,Z 219.864,A -85,B 0,C 180,E1 -28963.542,E2 -28963.542} C_VEL
LIN {X 0,Y 155.025,Z 210.644,A -85,B 0,C 180,E1 -28963.956,E2 -28963.956} C_VEL
LIN {X 0,Y 154.675,Z 206.123,A -85,B 0,C 180,E1 -28967.035,E2 -28967.035} C_VEL
LIN {X 0,Y 154.436,Z 204.536,A -85,B 0,C 180,E1 -28968.682,E2 -28968.682} C_VEL
LIN {X 0,Y 154.139,Z 202.576,A -85,B 0,C 180,E1 -28971.478,E2 -28971.478} C_VEL
LIN {X 0,Y 153.898,Z 202.024,A -85,B 0,C 180,E1 -28977.382,E2 -28977.382} C_VEL
LIN {X 0,Y 154.082,Z 202.551,A -85,B 0,C 180,E1 -28979.673,E2 -28979.673} C_VEL
LIN {X 0,Y 154.549,Z 205.688,A -85,B 0,C 180,E1 -28983.911,E2 -28983.911} C_VEL
LIN {X 0,Y 155.028,Z 208.669,A -85,B 0,C 180,E1 -28986.812,E2 -28986.812} C_VEL
LIN {X 0,Y 155.034,Z 208.872,A -85,B 0,C 180,E1 -28986.937,E2 -28986.937} C_VEL
LIN {X 0,Y 150.796,Z 221.957,A -85,B 0,C 180,E1 -28987.732,E2 -28987.732} C_VEL
LIN {X 0,Y 150.573,Z 222.511,A -85,B 0,C 180,E1 -28987.777,E2 -28987.777} C_VEL
LIN {X 0,Y 148.163,Z 227.989,A -85,B 0,C 180,E1 -28987.964,E2 -28987.964} C_VEL
LIN {X 0,Y 141.232,Z 239.96,A -85,B 0,C 180,E1 -28987.39,E2 -28987.39} C_VEL
LIN {X 0,Y 136.803,Z 246.485,A -85,B 0,C 180,E1 -28987.278,E2 -28987.278} C_VEL
LIN {X 0,Y 134.575,Z 249.605,A -85,B 0,C 180,E1 -28987.524,E2 -28987.524} C_VEL
LIN {X 0,Y 127.994,Z 258.085,A -85,B 0,C 180,E1 -28988.749,E2 -28988.749} C_VEL
LIN {X 0,Y 119.767,Z 266.997,A -85,B 0,C 180,E1 -28990.609,E2 -28990.609} C_VEL
LIN {X 0,Y 111.622,Z 274.301,A -85,B 0,C 180,E1 -28992.6,E2 -28992.6} C_VEL
LIN {X 0,Y 102.067,Z 281.426,A -85,B 0,C 180,E1 -28995.422,E2 -28995.422} C_VEL
LIN {X 0,Y 92.79,Z 287.058,A -85,B 0,C 180,E1 -28998.781,E2 -28998.781} C_VEL
LIN {X 0,Y 83.876,Z 291.45,A -85,B 0,C 180,E1 -29002.825,E2 -29002.825} C_VEL
LIN {X 0,Y 75.617,Z 294.683,A -85,B 0,C 180,E1 -29007.691,E2 -29007.691} C_VEL
LIN {X 0,Y 67.709,Z 296.993,A -85,B 0,C 180,E1 -29013.863,E2 -29013.863} C_VEL
LIN {X 0,Y 58.875,Z 298.514,A -85,B 0,C 180,E1 -29024.256,E2 -29024.256} C_VEL
LIN {X 0,Y 55.279,Z 298.675,A -85,B 0,C 180,E1 -29030.529,E2 -29030.529} C_VEL
LIN {X 0,Y 52.357,Z 298.396,A -85,B 0,C 180,E1 -29037.526,E2 -29037.526} C_VEL
LIN {X 0,Y 48.96,Z 296.666,A -85,B 0,C 180,E1 -29053.317,E2 -29053.317} C_VEL
LIN {X 0,Y 49.21,Z 293.617,A -85,B 0,C 180,E1 -29068.576,E2 -29068.576} C_VEL
LIN {X 0,Y 51.536,Z 289.547,A -85,B 0,C 180,E1 -29081.804,E2 -29081.804} C_VEL
LIN {X 0,Y 55.497,Z 284.744,A -85,B 0,C 180,E1 -29092.329,E2 -29092.329} C_VEL
LIN {X 0,Y 60.798,Z 278.702,A -85,B 0,C 180,E1 -29101.345,E2 -29101.345} C_VEL
LIN {X 0,Y 67.361,Z 271.178,A -85,B 0,C 180,E1 -29108.756,E2 -29108.756} C_VEL
LIN {X 0,Y 73.465,Z 263.498,A -85,B 0,C 180,E1 -29113.914,E2 -29113.914} C_VEL
LIN {X 0,Y 80.029,Z 254.138,A -85,B 0,C 180,E1 -29118.285,E2 -29118.285} C_VEL
LIN {X 0,Y 86.352,Z 243.708,A -85,B 0,C 180,E1 -29121.57,E2 -29121.57} C_VEL
LIN {X 0,Y 92.116,Z 232.133,A -85,B 0,C 180,E1 -29124.159,E2 -29124.159} C_VEL
LIN {X 0,Y 96.788,Z 219.923,A -85,B 0,C 180,E1 -29126.152,E2 -29126.152} C_VEL
LIN {X 0,Y 100.497,Z 206.46,A -85,B 0,C 180,E1 -29127.736,E2 -29127.736} C_VEL
LIN {X 0,Y 102.754,Z 194.151,A -85,B 0,C 180,E1 -29128.665,E2 -29128.665} C_VEL
LIN {X 0,Y 105.163,Z 171.704,A -85,B 0,C 180,E1 -29129.603,E2 -29129.603} C_VEL
LIN {X 0,Y 104.976,Z 170.594,A -85,B 0,C 180,E1 -29130.004,E2 -29130.004} C_VEL
LIN {X 0,Y 102.449,Z 164.277,A -85,B 0,C 180,E1 -29134.557,E2 -29134.557} C_VEL
LIN {X 0,Y 100.56,Z 160.122,A -85,B 0,C 180,E1 -29138.816,E2 -29138.816} C_VEL
LIN {X 0,Y 99.454,Z 157.702,A -85,B 0,C 180,E1 -29142.044,E2 -29142.044} C_VEL
LIN {X 0,Y 98.223,Z 154.445,A -85,B 0,C 180,E1 -29147.605,E2 -29147.605} C_VEL
LIN {X 0,Y 97.631,Z 153.552,A -85,B 0,C 180,E1 -29155.872,E2 -29155.872} C_VEL
LIN {X 0,Y 98.214,Z 154.166,A -85,B 0,C 180,E1 -29161.444,E2 -29161.444} C_VEL
LIN {X 0,Y 99.965,Z 158.567,A -85,B 0,C 180,E1 -29168.72,E2 -29168.72} C_VEL
LIN {X 0,Y 101.587,Z 162.305,A -85,B 0,C 180,E1 -29172.867,E2 -29172.867} C_VEL
LIN {X 0,Y 103.542,Z 166.864,A -85,B 0,C 180,E1 -29176.767,E2 -29176.767} C_VEL
LIN {X 0,Y 104.328,Z 169.155,A -85,B 0,C 180,E1 -29178.202,E2 -29178.202} C_VEL
LIN {X 0,Y 105.06,Z 173.071,A -85,B 0,C 180,E1 -29179.736,E2 -29179.736} C_VEL
LIN {X 0,Y 101.965,Z 201.002,A -85,B 0,C 180,E1 -29180.925,E2 -29180.925} C_VEL
LIN {X 0,Y 99.065,Z 214.637,A -85,B 0,C 180,E1 -29181.862,E2 -29181.862} C_VEL
LIN {X 0,Y 95.136,Z 227.199,A -85,B 0,C 180,E1 -29183.247,E2 -29183.247} C_VEL
LIN {X 0,Y 90.141,Z 238.921,A -85,B 0,C 180,E1 -29184.991,E2 -29184.991} C_VEL
LIN {X 0,Y 84.286,Z 250.299,A -85,B 0,C 180,E1 -29187.631,E2 -29187.631} C_VEL
LIN {X 0,Y 77.735,Z 260.459,A -85,B 0,C 180,E1 -29190.806,E2 -29190.806} C_VEL
LIN {X 0,Y 71.164,Z 269.701,A -85,B 0,C 180,E1 -29195.435,E2 -29195.435} C_VEL
LIN {X 0,Y 64.854,Z 277.271,A -85,B 0,C 180,E1 -29200.661,E2 -29200.661} C_VEL
LIN {X 0,Y 58.518,Z 284.748,A -85,B 0,C 180,E1 -29208.657,E2 -29208.657} C_VEL
LIN {X 0,Y 53.449,Z 290.726,A -85,B 0,C 180,E1 -29218.266,E2 -29218.266} C_VEL
LIN {X 0,Y 50.084,Z 295.427,A -85,B 0,C 180,E1 -29229.462,E2 -29229.462} C_VEL
LIN {X 0,Y 48.756,Z 298.994,A -85,B 0,C 180,E1 -29241.711,E2 -29241.711} C_VEL
LIN {X 0,Y 48.877,Z 300.781,A -85,B 0,C 180,E1 -29249.999,E2 -29249.999} C_VEL
LIN {X 0,Y 48.868,Z 302.055,A -85,B 0,C 180,E1 -29258.268,E2 -29258.268} C_VEL
LIN {X 0,Y 51.171,Z 303.406,A -85,B 0,C 180,E1 -29274.332,E2 -29274.332} C_VEL
LIN {X 0,Y 53.652,Z 303.489,A -85,B 0,C 180,E1 -29281.599,E2 -29281.599} C_VEL
LIN {X 0,Y 61.024,Z 302.484,A -85,B 0,C 180,E1 -29293.71,E2 -29293.71} C_VEL
LIN {X 0,Y 70.515,Z 299.952,A -85,B 0,C 180,E1 -29302.876,E2 -29302.876} C_VEL
LIN {X 0,Y 78.571,Z 296.943,A -85,B 0,C 180,E1 -29308.184,E2 -29308.184} C_VEL
LIN {X 0,Y 87.187,Z 292.92,A -85,B 0,C 180,E1 -29312.461,E2 -29312.461} C_VEL
LIN {X 0,Y 97.826,Z 286.793,A -85,B 0,C 180,E1 -29316.346,E2 -29316.346} C_VEL
LIN {X 0,Y 107.275,Z 280.132,A -85,B 0,C 180,E1 -29319,E2 -29319} C_VEL
LIN {X 0,Y 116.941,Z 271.893,A -85,B 0,C 180,E1 -29321.183,E2 -29321.183} C_VEL
LIN {X 0,Y 125.126,Z 263.488,A -85,B 0,C 180,E1 -29322.718,E2 -29322.718} C_VEL
LIN {X 0,Y 133.435,Z 253.136,A -85,B 0,C 180,E1 -29323.993,E2 -29323.993} C_VEL
LIN {X 0,Y 140.963,Z 241.495,A -85,B 0,C 180,E1 -29325.013,E2 -29325.013} C_VEL
LIN {X 0,Y 146.644,Z 230.44,A -85,B 0,C 180,E1 -29325.692,E2 -29325.692} C_VEL
LIN {X 0,Y 151.271,Z 218.727,A -85,B 0,C 180,E1 -29326.208,E2 -29326.208} C_VEL
LIN {X 0,Y 152.468,Z 215.061,A -85,B 0,C 180,E1 -29326.336,E2 -29326.336} C_VEL
LIN {X 0,Y 152.602,Z 213.568,A -85,B 0,C 180,E1 -29327.11,E2 -29327.11} C_VEL
LIN {X 0,Y 152.514,Z 211.224,A -85,B 0,C 180,E1 -29329.21,E2 -29329.21} C_VEL
LIN {X 0,Y 152.349,Z 209.344,A -85,B 0,C 180,E1 -29332.045,E2 -29332.045} C_VEL
LIN {X 0,Y 152.169,Z 208.894,A -85,B 0,C 180,E1 -29337.352,E2 -29337.352} C_VEL
LIN {X 0,Y 152.259,Z 209.302,A -85,B 0,C 180,E1 -29339.173,E2 -29339.173} C_VEL
LIN {X 0,Y 152.399,Z 211.656,A -85,B 0,C 180,E1 -29342.643,E2 -29342.643} C_VEL
LIN {X 0,Y 152.482,Z 213.289,A -85,B 0,C 180,E1 -29344.406,E2 -29344.406} C_VEL
LIN {X 0,Y 152.091,Z 214.698,A -85,B 0,C 180,E1 -29344.631,E2 -29344.631} C_VEL
LIN {X 0,Y 147.601,Z 226.627,A -85,B 0,C 180,E1 -29345.385,E2 -29345.385} C_VEL
LIN {X 0,Y 142.055,Z 237.833,A -85,B 0,C 180,E1 -29346.284,E2 -29346.284} C_VEL
LIN {X 0,Y 134.686,Z 249.447,A -85,B 0,C 180,E1 -29347.505,E2 -29347.505} C_VEL
LIN {X 0,Y 134.575,Z 249.605,A -85,B 0,C 180,E1 -29347.524,E2 -29347.524} C_VEL
LIN {X 0,Y 131.011,Z 254.259,A -85,B 0,C 180,E1 -29347.875,E2 -29347.875} C_VEL
LIN {X 0,Y 124.331,Z 261.592,A -85,B 0,C 180,E1 -29347.801,E2 -29347.801} C_VEL
LIN {X 0,Y 117.126,Z 268.373,A -85,B 0,C 180,E1 -29347.815,E2 -29347.815} C_VEL
LIN {X 0,Y 112.747,Z 272.152,A -85,B 0,C 180,E1 -29348.386,E2 -29348.386} C_VEL
LIN {X 0,Y 103.649,Z 279.196,A -85,B 0,C 180,E1 -29350.522,E2 -29350.522} C_VEL
LIN {X 0,Y 93.905,Z 285.378,A -85,B 0,C 180,E1 -29353.36,E2 -29353.36} C_VEL
LIN {X 0,Y 84.422,Z 290.244,A -85,B 0,C 180,E1 -29356.792,E2 -29356.792} C_VEL
LIN {X 0,Y 75.297,Z 293.951,A -85,B 0,C 180,E1 -29361.034,E2 -29361.034} C_VEL
LIN {X 0,Y 69.487,Z 295.843,A -85,B 0,C 180,E1 -29364.457,E2 -29364.457} C_VEL
LIN {X 0,Y 63.95,Z 297.283,A -85,B 0,C 180,E1 -29368.455,E2 -29368.455} C_VEL
LIN {X 0,Y 54.057,Z 298.863,A -85,B 0,C 180,E1 -29378.734,E2 -29378.734} C_VEL
LIN {X 0,Y 49.901,Z 299.063,A -85,B 0,C 180,E1 -29385.236,E2 -29385.236} C_VEL
LIN {X 0,Y 46.416,Z 298.832,A -85,B 0,C 180,E1 -29392.725,E2 -29392.725} C_VEL
LIN {X 0,Y 42.115,Z 297.158,A -85,B 0,C 180,E1 -29410.504,E2 -29410.504} C_VEL
LIN {X 0,Y 41.585,Z 295.724,A -85,B 0,C 180,E1 -29420.271,E2 -29420.271} C_VEL
LIN {X 0,Y 42.826,Z 292.735,A -85,B 0,C 180,E1 -29434.707,E2 -29434.707} C_VEL
LIN {X 0,Y 45.844,Z 288.756,A -85,B 0,C 180,E1 -29447.856,E2 -29447.856} C_VEL
LIN {X 0,Y 51.805,Z 282.63,A -85,B 0,C 180,E1 -29460.581,E2 -29460.581} C_VEL
LIN {X 0,Y 58.318,Z 275.963,A -85,B 0,C 180,E1 -29469.249,E2 -29469.249} C_VEL
LIN {X 0,Y 65.868,Z 267.685,A -85,B 0,C 180,E1 -29476.073,E2 -29476.073} C_VEL
LIN {X 0,Y 72.649,Z 259.187,A -85,B 0,C 180,E1 -29480.708,E2 -29480.708} C_VEL
LIN {X 0,Y 79.907,Z 248.661,A -85,B 0,C 180,E1 -29484.447,E2 -29484.447} C_VEL
LIN {X 0,Y 85.902,Z 238.229,A -85,B 0,C 180,E1 -29486.994,E2 -29486.994} C_VEL
LIN {X 0,Y 91.163,Z 226.803,A -85,B 0,C 180,E1 -29489.056,E2 -29489.056} C_VEL
LIN {X 0,Y 95.3,Z 215.011,A -85,B 0,C 180,E1 -29490.591,E2 -29490.591} C_VEL
LIN {X 0,Y 98.562,Z 201.792,A -85,B 0,C 180,E1 -29491.842,E2 -29491.842} C_VEL
LIN {X 0,Y 100.53,Z 188.978,A -85,B 0,C 180,E1 -29492.564,E2 -29492.564} C_VEL
LIN {X 0,Y 102.062,Z 174.572,A -85,B 0,C 180,E1 -29493.111,E2 -29493.111} C_VEL
LIN {X 0,Y 100.158,Z 169.331,A -85,B 0,C 180,E1 -29497.299,E2 -29497.299} C_VEL
LIN {X 0,Y 98.675,Z 165.666,A -85,B 0,C 180,E1 -29501.455,E2 -29501.455} C_VEL
LIN {X 0,Y 98.075,Z 164.198,A -85,B 0,C 180,E1 -29503.611,E2 -29503.611} C_VEL
LIN {X 0,Y 97.112,Z 161.224,A -85,B 0,C 180,E1 -29509.049,E2 -29509.049} C_VEL
LIN {X 0,Y 96.761,Z 160.58,A -85,B 0,C 180,E1 -29515.835,E2 -29515.835} C_VEL
LIN {X 0,Y 97.258,Z 161.207,A -85,B 0,C 180,E1 -29521.036,E2 -29521.036} C_VEL
LIN {X 0,Y 98.567,Z 165.156,A -85,B 0,C 180,E1 -29527.356,E2 -29527.356} C_VEL
LIN {X 0,Y 100.02,Z 168.928,A -85,B 0,C 180,E1 -29531.591,E2 -29531.591} C_VEL
LIN {X 0,Y 101.722,Z 173.494,A -85,B 0,C 180,E1 -29535.426,E2 -29535.426} C_VEL
LIN {X 0,Y 102.032,Z 175.172,A -85,B 0,C 180,E1 -29536.202,E2 -29536.202} C_VEL
LIN {X 0,Y 99.055,Z 200.765,A -85,B 0,C 180,E1 -29537.237,E2 -29537.237} C_VEL
LIN {X 0,Y 96.098,Z 214.137,A -85,B 0,C 180,E1 -29538.057,E2 -29538.057} C_VEL
LIN {X 0,Y 92.156,Z 226.438,A -85,B 0,C 180,E1 -29539.308,E2 -29539.308} C_VEL
LIN {X 0,Y 87.374,Z 237.444,A -85,B 0,C 180,E1 -29540.759,E2 -29540.759} C_VEL
LIN {X 0,Y 81.96,Z 247.7,A -85,B 0,C 180,E1 -29542.807,E2 -29542.807} C_VEL
LIN {X 0,Y 75.107,Z 258.313,A -85,B 0,C 180,E1 -29545.755,E2 -29545.755} C_VEL
LIN {X 0,Y 68.656,Z 267.024,A -85,B 0,C 180,E1 -29549.527,E2 -29549.527} C_VEL
LIN {X 0,Y 61.831,Z 275.026,A -85,B 0,C 180,E1 -29554.505,E2 -29554.505} C_VEL
LIN {X 0,Y 57.082,Z 279.987,A -85,B 0,C 180,E1 -29558.797,E2 -29558.797} C_VEL
LIN {X 0,Y 50.29,Z 287.177,A -85,B 0,C 180,E1 -29568.408,E2 -29568.408} C_VEL
LIN {X 0,Y 44.598,Z 293.347,A -85,B 0,C 180,E1 -29581.785,E2 -29581.785} C_VEL
LIN {X 0,Y 42.039,Z 297.344,A -85,B 0,C 180,E1 -29595.476,E2 -29595.476} C_VEL
LIN {X 0,Y 41.764,Z 300.27,A -85,B 0,C 180,E1 -29609.999,E2 -29609.999} C_VEL
LIN {X 0,Y 41.84,Z 301.573,A -85,B 0,C 180,E1 -29619.669,E2 -29619.669} C_VEL
LIN {X 0,Y 44.756,Z 302.977,A -85,B 0,C 180,E1 -29638.105,E2 -29638.105} C_VEL
LIN {X 0,Y 47.72,Z 303.109,A -85,B 0,C 180,E1 -29646.093,E2 -29646.093} C_VEL
LIN {X 0,Y 56.081,Z 302.167,A -85,B 0,C 180,E1 -29658.756,E2 -29658.756} C_VEL
LIN {X 0,Y 66.456,Z 299.702,A -85,B 0,C 180,E1 -29667.783,E2 -29667.783} C_VEL
LIN {X 0,Y 75.055,Z 296.742,A -85,B 0,C 180,E1 -29672.818,E2 -29672.818} C_VEL
LIN {X 0,Y 84.132,Z 292.78,A -85,B 0,C 180,E1 -29676.764,E2 -29676.764} C_VEL
LIN {X 0,Y 93.595,Z 287.716,A -85,B 0,C 180,E1 -29679.821,E2 -29679.821} C_VEL
LIN {X 0,Y 103.294,Z 281.393,A -85,B 0,C 180,E1 -29682.278,E2 -29682.278} C_VEL
LIN {X 0,Y 113.19,Z 273.508,A -85,B 0,C 180,E1 -29684.238,E2 -29684.238} C_VEL
LIN {X 0,Y 123.207,Z 263.717,A -85,B 0,C 180,E1 -29685.864,E2 -29685.864} C_VEL
LIN {X 0,Y 131.659,Z 253.558,A -85,B 0,C 180,E1 -29686.955,E2 -29686.955} C_VEL
LIN {X 0,Y 138.449,Z 243.514,A -85,B 0,C 180,E1 -29687.737,E2 -29687.737} C_VEL
LIN {X 0,Y 144.846,Z 231.716,A -85,B 0,C 180,E1 -29688.379,E2 -29688.379} C_VEL
LIN {X 0,Y 149.625,Z 220.337,A -85,B 0,C 180,E1 -29688.829,E2 -29688.829} C_VEL
LIN {X 0,Y 150.238,Z 218.47,A -85,B 0,C 180,E1 -29689.045,E2 -29689.045} C_VEL
LIN {X 0,Y 150.216,Z 216.321,A -85,B 0,C 180,E1 -29691.931,E2 -29691.931} C_VEL
LIN {X 0,Y 150.073,Z 215.656,A -85,B 0,C 180,E1 -29697.315,E2 -29697.315} C_VEL
LIN {X 0,Y 149.997,Z 217.686,A -85,B 0,C 180,E1 -29701.343,E2 -29701.343} C_VEL
LIN {X 0,Y 149.991,Z 218.197,A -85,B 0,C 180,E1 -29702.081,E2 -29702.081} C_VEL
LIN {X 0,Y 145.212,Z 229.753,A -85,B 0,C 180,E1 -29702.843,E2 -29702.843} C_VEL
LIN {X 0,Y 139.094,Z 241.138,A -85,B 0,C 180,E1 -29703.703,E2 -29703.703} C_VEL
LIN {X 0,Y 132.219,Z 251.362,A -85,B 0,C 180,E1 -29704.694,E2 -29704.694} C_VEL
LIN {X 0,Y 124.295,Z 260.976,A -85,B 0,C 180,E1 -29706.037,E2 -29706.037} C_VEL
LIN {X 0,Y 115.288,Z 269.926,A -85,B 0,C 180,E1 -29707.858,E2 -29707.858} C_VEL
LIN {X 0,Y 112.747,Z 272.152,A -85,B 0,C 180,E1 -29708.386,E2 -29708.386} C_VEL
LIN {X 0,Y 108.198,Z 275.764,A -85,B 0,C 180,E1 -29709.034,E2 -29709.034} C_VEL
LIN {X 0,Y 96.549,Z 283.295,A -85,B 0,C 180,E1 -29709.398,E2 -29709.398} C_VEL
LIN {X 0,Y 89.653,Z 287.024,A -85,B 0,C 180,E1 -29709.995,E2 -29709.995} C_VEL
LIN {X 0,Y 86.305,Z 288.662,A -85,B 0,C 180,E1 -29710.763,E2 -29710.763} C_VEL
LIN {X 0,Y 76.17,Z 293.02,A -85,B 0,C 180,E1 -29714.349,E2 -29714.349} C_VEL
LIN {X 0,Y 66.808,Z 296.073,A -85,B 0,C 180,E1 -29718.777,E2 -29718.777} C_VEL
LIN {X 0,Y 60.825,Z 297.567,A -85,B 0,C 180,E1 -29722.428,E2 -29722.428} C_VEL
LIN {X 0,Y 55.142,Z 298.591,A -85,B 0,C 180,E1 -29726.854,E2 -29726.854} C_VEL
LIN {X 0,Y 45.056,Z 299.44,A -85,B 0,C 180,E1 -29738.747,E2 -29738.747} C_VEL
LIN {X 0,Y 40.884,Z 299.267,A -85,B 0,C 180,E1 -29746.56,E2 -29746.56} C_VEL
LIN {X 0,Y 35.382,Z 297.652,A -85,B 0,C 180,E1 -29766.593,E2 -29766.593} C_VEL
LIN {X 0,Y 34.508,Z 296.249,A -85,B 0,C 180,E1 -29778.25,E2 -29778.25} C_VEL
LIN {X 0,Y 35.454,Z 293.659,A -85,B 0,C 180,E1 -29793.878,E2 -29793.878} C_VEL
LIN {X 0,Y 39.136,Z 289.396,A -85,B 0,C 180,E1 -29811.049,E2 -29811.049} C_VEL
LIN {X 0,Y 44.748,Z 284.346,A -85,B 0,C 180,E1 -29823.348,E2 -29823.348} C_VEL
LIN {X 0,Y 51.728,Z 278.016,A -85,B 0,C 180,E1 -29832.792,E2 -29832.792} C_VEL
LIN {X 0,Y 59.769,Z 270.082,A -85,B 0,C 180,E1 -29839.847,E2 -29839.847} C_VEL
LIN {X 0,Y 68.392,Z 260.234,A -85,B 0,C 180,E1 -29845.295,E2 -29845.295} C_VEL
LIN {X 0,Y 75.265,Z 251.044,A -85,B 0,C 180,E1 -29848.438,E2 -29848.438} C_VEL
LIN {X 0,Y 82.262,Z 239.63,A -85,B 0,C 180,E1 -29851.13,E2 -29851.13} C_VEL
LIN {X 0,Y 87.753,Z 228.453,A -85,B 0,C 180,E1 -29852.999,E2 -29852.999} C_VEL
LIN {X 0,Y 92.45,Z 215.942,A -85,B 0,C 180,E1 -29854.521,E2 -29854.521} C_VEL
LIN {X 0,Y 95.78,Z 203.252,A -85,B 0,C 180,E1 -29855.655,E2 -29855.655} C_VEL
LIN {X 0,Y 98.04,Z 189.514,A -85,B 0,C 180,E1 -29856.387,E2 -29856.387} C_VEL
LIN {X 0,Y 99.286,Z 178.124,A -85,B 0,C 180,E1 -29856.809,E2 -29856.809} C_VEL
LIN {X 0,Y 97.844,Z 173.637,A -85,B 0,C 180,E1 -29861.006,E2 -29861.006} C_VEL
LIN {X 0,Y 96.874,Z 170.927,A -85,B 0,C 180,E1 -29864.753,E2 -29864.753} C_VEL
LIN {X 0,Y 96.144,Z 168.187,A -85,B 0,C 180,E1 -29869.737,E2 -29869.737} C_VEL
LIN {X 0,Y 95.888,Z 167.637,A -85,B 0,C 180,E1 -29875.797,E2 -29875.797} C_VEL
LIN {X 0,Y 96.23,Z 168.044,A -85,B 0,C 180,E1 -29880.001,E2 -29880.001} C_VEL
LIN {X 0,Y 97.294,Z 171.948,A -85,B 0,C 180,E1 -29886.221,E2 -29886.221} C_VEL
LIN {X 0,Y 98.549,Z 175.665,A -85,B 0,C 180,E1 -29890.4,E2 -29890.4} C_VEL
LIN {X 0,Y 99.327,Z 178.144,A -85,B 0,C 180,E1 -29892.515,E2 -29892.515} C_VEL
LIN {X 0,Y 96.69,Z 199.922,A -85,B 0,C 180,E1 -29893.322,E2 -29893.322} C_VEL
LIN {X 0,Y 93.726,Z 213.186,A -85,B 0,C 180,E1 -29894.041,E2 -29894.041} C_VEL
LIN {X 0,Y 89.64,Z 225.674,A -85,B 0,C 180,E1 -29895.128,E2 -29895.128} C_VEL
LIN {X 0,Y 84.293,Z 237.557,A -85,B 0,C 180,E1 -29896.496,E2 -29896.496} C_VEL
LIN {X 0,Y 78.664,Z 247.722,A -85,B 0,C 180,E1 -29898.327,E2 -29898.327} C_VEL
LIN {X 0,Y 71.508,Z 258.266,A -85,B 0,C 180,E1 -29900.981,E2 -29900.981} C_VEL
LIN {X 0,Y 63.933,Z 267.795,A -85,B 0,C 180,E1 -29904.918,E2 -29904.918} C_VEL
LIN {X 0,Y 56.001,Z 276.161,A -85,B 0,C 180,E1 -29910.133,E2 -29910.133} C_VEL
LIN {X 0,Y 49.937,Z 282.061,A -85,B 0,C 180,E1 -29915.977,E2 -29915.977} C_VEL
LIN {X 0,Y 44.092,Z 287.466,A -85,B 0,C 180,E1 -29924.169,E2 -29924.169} C_VEL
LIN {X 0,Y 38.443,Z 292.706,A -85,B 0,C 180,E1 -29936.738,E2 -29936.738} C_VEL
LIN {X 0,Y 35.181,Z 296.768,A -85,B 0,C 180,E1 -29952.562,E2 -29952.562} C_VEL
LIN {X 0,Y 34.662,Z 299.747,A -85,B 0,C 180,E1 -29969.999,E2 -29969.999} C_VEL
LIN {X 0,Y 34.845,Z 301.09,A -85,B 0,C 180,E1 -29981.635,E2 -29981.635} C_VEL
LIN {X 0,Y 38.604,Z 302.549,A -85,B 0,C 180,E1 -30003.103,E2 -30003.103} C_VEL
LIN {X 0,Y 42.166,Z 302.714,A -85,B 0,C 180,E1 -30011.812,E2 -30011.812} C_VEL
LIN {X 0,Y 46.626,Z 302.484,A -85,B 0,C 180,E1 -30018.908,E2 -30018.908} C_VEL
LIN {X 0,Y 57.162,Z 300.839,A -85,B 0,C 180,E1 -30029.388,E2 -30029.388} C_VEL
LIN {X 0,Y 64.277,Z 299.076,A -85,B 0,C 180,E1 -30034.064,E2 -30034.064} C_VEL
LIN {X 0,Y 75.211,Z 295.352,A -85,B 0,C 180,E1 -30039.137,E2 -30039.137} C_VEL
LIN {X 0,Y 84.824,Z 291.101,A -85,B 0,C 180,E1 -30042.33,E2 -30042.33} C_VEL
LIN {X 0,Y 96.367,Z 284.687,A -85,B 0,C 180,E1 -30045.087,E2 -30045.087} C_VEL
LIN {X 0,Y 106.399,Z 277.733,A -85,B 0,C 180,E1 -30046.978,E2 -30046.978} C_VEL
LIN {X 0,Y 116.569,Z 269.052,A -85,B 0,C 180,E1 -30048.443,E2 -30048.443} C_VEL
LIN {X 0,Y 125.114,Z 260.18,A -85,B 0,C 180,E1 -30049.429,E2 -30049.429} C_VEL
LIN {X 0,Y 133.671,Z 249.286,A -85,B 0,C 180,E1 -30050.34,E2 -30050.34} C_VEL
LIN {X 0,Y 140.577,Z 238.28,A -85,B 0,C 180,E1 -30050.889,E2 -30050.889} C_VEL
LIN {X 0,Y 146.45,Z 226.356,A -85,B 0,C 180,E1 -30051.358,E2 -30051.358} C_VEL
LIN {X 0,Y 147.651,Z 223.415,A -85,B 0,C 180,E1 -30051.609,E2 -30051.609} C_VEL
LIN {X 0,Y 147.559,Z 222.552,A -85,B 0,C 180,E1 -30054.534,E2 -30054.534} C_VEL
LIN {X 0,Y 147.591,Z 222.365,A -85,B 0,C 180,E1 -30057.27,E2 -30057.27} C_VEL
LIN {X 0,Y 147.411,Z 223.43,A -85,B 0,C 180,E1 -30059.659,E2 -30059.659} C_VEL
LIN {X 0,Y 141.621,Z 235.578,A -85,B 0,C 180,E1 -30060.374,E2 -30060.374} C_VEL
LIN {X 0,Y 134.443,Z 247.288,A -85,B 0,C 180,E1 -30061.252,E2 -30061.252} C_VEL
LIN {X 0,Y 126.602,Z 257.445,A -85,B 0,C 180,E1 -30062.254,E2 -30062.254} C_VEL
LIN {X 0,Y 117.162,Z 267.355,A -85,B 0,C 180,E1 -30063.789,E2 -30063.789} C_VEL
LIN {X 0,Y 107.671,Z 275.463,A -85,B 0,C 180,E1 -30065.49,E2 -30065.49} C_VEL
LIN {X 0,Y 97.405,Z 282.555,A -85,B 0,C 180,E1 -30067.728,E2 -30067.728} C_VEL
LIN {X 0,Y 86.305,Z 288.662,A -85,B 0,C 180,E1 -30070.763,E2 -30070.763} C_VEL
LIN {X 0,Y 81.144,Z 291.004,A -85,B 0,C 180,E1 -30071.932,E2 -30071.932} C_VEL
LIN {X 0,Y 71.912,Z 294.388,A -85,B 0,C 180,E1 -30072.982,E2 -30072.982} C_VEL
LIN {X 0,Y 62.496,Z 296.971,A -85,B 0,C 180,E1 -30074.43,E2 -30074.43} C_VEL
LIN {X 0,Y 57.136,Z 298.057,A -85,B 0,C 180,E1 -30076.564,E2 -30076.564} C_VEL
LIN {X 0,Y 46.375,Z 299.562,A -85,B 0,C 180,E1 -30084.593,E2 -30084.593} C_VEL
LIN {X 0,Y 40.399,Z 299.83,A -85,B 0,C 180,E1 -30091.458,E2 -30091.458} C_VEL
LIN {X 0,Y 31.848,Z 299.12,A -85,B 0,C 180,E1 -30108.546,E2 -30108.546} C_VEL
LIN {X 0,Y 27.49,Z 296.771,A -85,B 0,C 180,E1 -30135.189,E2 -30135.189} C_VEL
LIN {X 0,Y 28.153,Z 294.505,A -85,B 0,C 180,E1 -30153.113,E2 -30153.113} C_VEL
LIN {X 0,Y 30.995,Z 291.458,A -85,B 0,C 180,E1 -30169.885,E2 -30169.885} C_VEL
LIN {X 0,Y 36.735,Z 286.86,A -85,B 0,C 180,E1 -30185.028,E2 -30185.028} C_VEL
LIN {X 0,Y 45.401,Z 279.931,A -85,B 0,C 180,E1 -30197.333,E2 -30197.333} C_VEL
LIN {X 0,Y 53.974,Z 272.423,A -85,B 0,C 180,E1 -30204.472,E2 -30204.472} C_VEL
LIN {X 0,Y 61.532,Z 264.765,A -85,B 0,C 180,E1 -30208.942,E2 -30208.942} C_VEL
LIN {X 0,Y 69.369,Z 255.438,A -85,B 0,C 180,E1 -30212.437,E2 -30212.437} C_VEL
LIN {X 0,Y 76.648,Z 245.038,A -85,B 0,C 180,E1 -30214.887,E2 -30214.887} C_VEL
LIN {X 0,Y 83.179,Z 233.499,A -85,B 0,C 180,E1 -30216.761,E2 -30216.761} C_VEL
LIN {X 0,Y 88.439,Z 221.391,A -85,B 0,C 180,E1 -30218.247,E2 -30218.247} C_VEL
LIN {X 0,Y 92.551,Z 208.349,A -85,B 0,C 180,E1 -30219.423,E2 -30219.423} C_VEL
LIN {X 0,Y 95.287,Z 195.339,A -85,B 0,C 180,E1 -30220.18,E2 -30220.18} C_VEL
LIN {X 0,Y 96.918,Z 181.878,A -85,B 0,C 180,E1 -30220.711,E2 -30220.711} C_VEL
LIN {X 0,Y 95.817,Z 177.913,A -85,B 0,C 180,E1 -30225.401,E2 -30225.401} C_VEL
LIN {X 0,Y 95.188,Z 175.161,A -85,B 0,C 180,E1 -30230.438,E2 -30230.438} C_VEL
LIN {X 0,Y 95.014,Z 174.694,A -85,B 0,C 180,E1 -30235.759,E2 -30235.759} C_VEL
LIN {X 0,Y 95.247,Z 175.052,A -85,B 0,C 180,E1 -30239.208,E2 -30239.208} C_VEL
LIN {X 0,Y 96.02,Z 178.565,A -85,B 0,C 180,E1 -30244.855,E2 -30244.855} C_VEL
LIN {X 0,Y 96.943,Z 181.88,A -85,B 0,C 180,E1 -30248.599,E2 -30248.599} C_VEL
LIN {X 0,Y 94.509,Z 200.624,A -85,B 0,C 180,E1 -30249.274,E2 -30249.274} C_VEL
LIN {X 0,Y 91.355,Z 213.92,A -85,B 0,C 180,E1 -30249.889,E2 -30249.889} C_VEL
LIN {X 0,Y 87.461,Z 225.306,A -85,B 0,C 180,E1 -30250.763,E2 -30250.763} C_VEL
LIN {X 0,Y 82.558,Z 236.082,A -85,B 0,C 180,E1 -30251.765,E2 -30251.765} C_VEL
LIN {X 0,Y 75.887,Z 247.744,A -85,B 0,C 180,E1 -30253.484,E2 -30253.484} C_VEL
LIN {X 0,Y 68.456,Z 258.219,A -85,B 0,C 180,E1 -30255.743,E2 -30255.743} C_VEL
LIN {X 0,Y 61.263,Z 266.818,A -85,B 0,C 180,E1 -30258.835,E2 -30258.835} C_VEL
LIN {X 0,Y 53.469,Z 274.713,A -85,B 0,C 180,E1 -30263.059,E2 -30263.059} C_VEL
LIN {X 0,Y 47.465,Z 280.009,A -85,B 0,C 180,E1 -30267.325,E2 -30267.325} C_VEL
LIN {X 0,Y 39.427,Z 286.727,A -85,B 0,C 180,E1 -30276.664,E2 -30276.664} C_VEL
LIN {X 0,Y 32.685,Z 292.045,A -85,B 0,C 180,E1 -30289.828,E2 -30289.828} C_VEL
LIN {X 0,Y 28.442,Z 296.174,A -85,B 0,C 180,E1 -30308.243,E2 -30308.243} C_VEL
LIN {X 0,Y 27.551,Z 299.21,A -85,B 0,C 180,E1 -30329.999,E2 -30329.999} C_VEL
LIN {X 0,Y 27.901,Z 300.607,A -85,B 0,C 180,E1 -30344.588,E2 -30344.588} C_VEL
LIN {X 0,Y 32.863,Z 302.121,A -85,B 0,C 180,E1 -30369.908,E2 -30369.908} C_VEL
LIN {X 0,Y 42.281,Z 302.133,A -85,B 0,C 180,E1 -30386.212,E2 -30386.212} C_VEL
LIN {X 0,Y 53.879,Z 300.55,A -85,B 0,C 180,E1 -30395.934,E2 -30395.934} C_VEL
LIN {X 0,Y 60.787,Z 299.01,A -85,B 0,C 180,E1 -30399.704,E2 -30399.704} C_VEL
LIN {X 0,Y 69.707,Z 296.337,A -85,B 0,C 180,E1 -30403.297,E2 -30403.297} C_VEL
LIN {X 0,Y 79.597,Z 292.499,A -85,B 0,C 180,E1 -30406.225,E2 -30406.225} C_VEL
LIN {X 0,Y 89.692,Z 287.568,A -85,B 0,C 180,E1 -30408.369,E2 -30408.369} C_VEL
LIN {X 0,Y 99.89,Z 281.394,A -85,B 0,C 180,E1 -30410.065,E2 -30410.065} C_VEL
LIN {X 0,Y 110.19,Z 273.748,A -85,B 0,C 180,E1 -30411.341,E2 -30411.341} C_VEL
LIN {X 0,Y 120.53,Z 264.173,A -85,B 0,C 180,E1 -30412.42,E2 -30412.42} C_VEL
LIN {X 0,Y 128.338,Z 255.378,A -85,B 0,C 180,E1 -30413.004,E2 -30413.004} C_VEL
LIN {X 0,Y 136.145,Z 244.646,A -85,B 0,C 180,E1 -30413.574,E2 -30413.574} C_VEL
LIN {X 0,Y 142.283,Z 234.152,A -85,B 0,C 180,E1 -30413.917,E2 -30413.917} C_VEL
LIN {X 0,Y 143.838,Z 231.012,A -85,B 0,C 180,E1 -30414.01,E2 -30414.01} C_VEL
LIN {X 0,Y 144.735,Z 229.106,A -85,B 0,C 180,E1 -30414.427,E2 -30414.427} C_VEL
LIN {X 0,Y 144.32,Z 229.764,A -85,B 0,C 180,E1 -30417.208,E2 -30417.208} C_VEL
LIN {X 0,Y 138.024,Z 241.29,A -85,B 0,C 180,E1 -30417.826,E2 -30417.826} C_VEL
LIN {X 0,Y 130.941,Z 251.625,A -85,B 0,C 180,E1 -30418.517,E2 -30418.517} C_VEL
LIN {X 0,Y 122.997,Z 261.075,A -85,B 0,C 180,E1 -30419.402,E2 -30419.402} C_VEL
LIN {X 0,Y 113.874,Z 269.916,A -85,B 0,C 180,E1 -30420.669,E2 -30420.669} C_VEL
LIN {X 0,Y 103.738,Z 277.91,A -85,B 0,C 180,E1 -30422.177,E2 -30422.177} C_VEL
LIN {X 0,Y 92.148,Z 285.236,A -85,B 0,C 180,E1 -30424.374,E2 -30424.374} C_VEL
LIN {X 0,Y 81.419,Z 290.511,A -85,B 0,C 180,E1 -30426.941,E2 -30426.941} C_VEL
LIN {X 0,Y 71.382,Z 294.348,A -85,B 0,C 180,E1 -30430.079,E2 -30430.079} C_VEL
LIN {X 0,Y 64.833,Z 296.303,A -85,B 0,C 180,E1 -30432.681,E2 -30432.681} C_VEL
LIN {X 0,Y 57.136,Z 298.057,A -85,B 0,C 180,E1 -30436.564,E2 -30436.564} C_VEL
LIN {X 0,Y 51.817,Z 298.969,A -85,B 0,C 180,E1 -30439.148,E2 -30439.148} C_VEL
LIN {X 0,Y 42.374,Z 299.928,A -85,B 0,C 180,E1 -30442.703,E2 -30442.703} C_VEL
LIN {X 0,Y 34.877,Z 300.126,A -85,B 0,C 180,E1 -30446.677,E2 -30446.677} C_VEL
LIN {X 0,Y 29.82,Z 299.918,A -85,B 0,C 180,E1 -30452.163,E2 -30452.163} C_VEL
LIN {X 0,Y 28.376,Z 299.745,A -85,B 0,C 180,E1 -30454.808,E2 -30454.808} C_VEL
LIN {X 0,Y 22.866,Z 298.637,A -85,B 0,C 180,E1 -30472.071,E2 -30472.071} C_VEL
LIN {X 0,Y 20.603,Z 297.293,A -85,B 0,C 180,E1 -30490.057,E2 -30490.057} C_VEL
LIN {X 0,Y 21.224,Z 294.801,A -85,B 0,C 180,E1 -30516.615,E2 -30516.615} C_VEL
LIN {X 0,Y 26.376,Z 290.674,A -85,B 0,C 180,E1 -30542.204,E2 -30542.204} C_VEL
LIN {X 0,Y 33.813,Z 285.759,A -85,B 0,C 180,E1 -30556.678,E2 -30556.678} C_VEL
LIN {X 0,Y 42.438,Z 279.595,A -85,B 0,C 180,E1 -30565.899,E2 -30565.899} C_VEL
LIN {X 0,Y 51.775,Z 271.91,A -85,B 0,C 180,E1 -30571.926,E2 -30571.926} C_VEL
LIN {X 0,Y 61.457,Z 262.266,A -85,B 0,C 180,E1 -30576.187,E2 -30576.187} C_VEL
LIN {X 0,Y 68.906,Z 253.367,A -85,B 0,C 180,E1 -30578.546,E2 -30578.546} C_VEL
LIN {X 0,Y 76.439,Z 242.43,A -85,B 0,C 180,E1 -30580.462,E2 -30580.462} C_VEL
LIN {X 0,Y 82.325,Z 231.72,A -85,B 0,C 180,E1 -30581.758,E2 -30581.758} C_VEL
LIN {X 0,Y 87.747,Z 218.893,A -85,B 0,C 180,E1 -30582.967,E2 -30582.967} C_VEL
LIN {X 0,Y 91.615,Z 206.081,A -85,B 0,C 180,E1 -30583.889,E2 -30583.889} C_VEL
LIN {X 0,Y 93.993,Z 193.925,A -85,B 0,C 180,E1 -30584.443,E2 -30584.443} C_VEL
LIN {X 0,Y 94.968,Z 186.054,A -85,B 0,C 180,E1 -30584.782,E2 -30584.782} C_VEL
LIN {X 0,Y 94.435,Z 183.758,A -85,B 0,C 180,E1 -30588.327,E2 -30588.327} C_VEL
LIN {X 0,Y 94.226,Z 182.105,A -85,B 0,C 180,E1 -30591.421,E2 -30591.421} C_VEL
LIN {X 0,Y 94.143,Z 181.731,A -85,B 0,C 180,E1 -30595.719,E2 -30595.719} C_VEL
LIN {X 0,Y 94.282,Z 182.062,A -85,B 0,C 180,E1 -30598.399,E2 -30598.399} C_VEL
LIN {X 0,Y 94.803,Z 185.175,A -85,B 0,C 180,E1 -30603.454,E2 -30603.454} C_VEL
LIN {X 0,Y 94.99,Z 185.963,A -85,B 0,C 180,E1 -30604.508,E2 -30604.508} C_VEL
LIN {X 0,Y 92.844,Z 201.214,A -85,B 0,C 180,E1 -30605.062,E2 -30605.062} C_VEL
LIN {X 0,Y 89.656,Z 214.05,A -85,B 0,C 180,E1 -30605.534,E2 -30605.534} C_VEL
LIN {X 0,Y 84.856,Z 227.156,A -85,B 0,C 180,E1 -30606.338,E2 -30606.338} C_VEL
LIN {X 0,Y 78.817,Z 239.371,A -85,B 0,C 180,E1 -30607.246,E2 -30607.246} C_VEL
LIN {X 0,Y 72.001,Z 250.309,A -85,B 0,C 180,E1 -30608.768,E2 -30608.768} C_VEL
LIN {X 0,Y 64.333,Z 260.162,A -85,B 0,C 180,E1 -30610.511,E2 -30610.511} C_VEL
LIN {X 0,Y 56.032,Z 269.194,A -85,B 0,C 180,E1 -30613.568,E2 -30613.568} C_VEL
LIN {X 0,Y 47.455,Z 276.891,A -85,B 0,C 180,E1 -30617.355,E2 -30617.355} C_VEL
LIN {X 0,Y 38.519,Z 283.911,A -85,B 0,C 180,E1 -30624.173,E2 -30624.173} C_VEL
LIN {X 0,Y 30.1,Z 289.739,A -85,B 0,C 180,E1 -30635.192,E2 -30635.192} C_VEL
LIN {X 0,Y 23.467,Z 294.309,A -85,B 0,C 180,E1 -30653.201,E2 -30653.201} C_VEL
LIN {X 0,Y 20.936,Z 296.715,A -85,B 0,C 180,E1 -30670.384,E2 -30670.384} C_VEL
LIN {X 0,Y 20.439,Z 298.671,A -85,B 0,C 180,E1 -30689.998,E2 -30689.998} C_VEL
LIN {X 0,Y 21.09,Z 300.116,A -85,B 0,C 180,E1 -30709.464,E2 -30709.464} C_VEL
LIN {X 0,Y 27.779,Z 301.694,A -85,B 0,C 180,E1 -30739.375,E2 -30739.375} C_VEL
LIN {X 0,Y 38.772,Z 301.766,A -85,B 0,C 180,E1 -30755,E2 -30755} C_VEL
LIN {X 0,Y 44.951,Z 301.214,A -85,B 0,C 180,E1 -30759.732,E2 -30759.732} C_VEL
LIN {X 0,Y 57.954,Z 298.919,A -85,B 0,C 180,E1 -30765.963,E2 -30765.963} C_VEL
LIN {X 0,Y 68.003,Z 296.134,A -85,B 0,C 180,E1 -30769.055,E2 -30769.055} C_VEL
LIN {X 0,Y 78.209,Z 292.358,A -85,B 0,C 180,E1 -30771.295,E2 -30771.295} C_VEL
LIN {X 0,Y 88.535,Z 287.494,A -85,B 0,C 180,E1 -30772.871,E2 -30772.871} C_VEL
LIN {X 0,Y 98.913,Z 281.392,A -85,B 0,C 180,E1 -30774.117,E2 -30774.117} C_VEL
LIN {X 0,Y 109.348,Z 273.834,A -85,B 0,C 180,E1 -30775.016,E2 -30775.016} C_VEL
LIN {X 0,Y 118.035,Z 266.163,A -85,B 0,C 180,E1 -30775.658,E2 -30775.658} C_VEL
LIN {X 0,Y 119.8,Z 264.401,A -85,B 0,C 180,E1 -30775.786,E2 -30775.786} C_VEL
LIN {X 0,Y 119.713,Z 264.442,A -85,B 0,C 180,E1 -30776.397,E2 -30776.397} C_VEL
LIN {X 0,Y 110.808,Z 272.477,A -85,B 0,C 180,E1 -30777.372,E2 -30777.372} C_VEL
LIN {X 0,Y 100.178,Z 280.275,A -85,B 0,C 180,E1 -30778.625,E2 -30778.625} C_VEL
LIN {X 0,Y 91.009,Z 285.749,A -85,B 0,C 180,E1 -30779.999,E2 -30779.999} C_VEL
LIN {X 0,Y 80.864,Z 290.643,A -85,B 0,C 180,E1 -30781.839,E2 -30781.839} C_VEL
LIN {X 0,Y 70.474,Z 294.547,A -85,B 0,C 180,E1 -30784.253,E2 -30784.253} C_VEL
LIN {X 0,Y 63.491,Z 296.571,A -85,B 0,C 180,E1 -30786.355,E2 -30786.355} C_VEL
LIN {X 0,Y 54.039,Z 298.581,A -85,B 0,C 180,E1 -30790.013,E2 -30790.013} C_VEL
LIN {X 0,Y 43.848,Z 299.912,A -85,B 0,C 180,E1 -30795.911,E2 -30795.911} C_VEL
LIN {X 0,Y 36.234,Z 300.225,A -85,B 0,C 180,E1 -30802.824,E2 -30802.824} C_VEL
LIN {X 0,Y 28.376,Z 299.745,A -85,B 0,C 180,E1 -30814.808,E2 -30814.808} C_VEL
LIN {X 0,Y 24.172,Z 299.207,A -85,B 0,C 180,E1 -30823.809,E2 -30823.809} C_VEL
LIN {X 0,Y 17.528,Z 297.778,A -85,B 0,C 180,E1 -30843.978,E2 -30843.978} C_VEL
LIN {X 0,Y 14.647,Z 296.062,A -85,B 0,C 180,E1 -30870.095,E2 -30870.095} C_VEL
LIN {X 0,Y 15.529,Z 294.378,A -85,B 0,C 180,E1 -30891.639,E2 -30891.639} C_VEL
LIN {X 0,Y 16.445,Z 293.734,A -85,B 0,C 180,E1 -30897.509,E2 -30897.509} C_VEL
LIN {X 0,Y 23.436,Z 289.85,A -85,B 0,C 180,E1 -30918.567,E2 -30918.567} C_VEL
LIN {X 0,Y 34.1,Z 283.587,A -85,B 0,C 180,E1 -30931.156,E2 -30931.156} C_VEL
LIN {X 0,Y 43.849,Z 276.79,A -85,B 0,C 180,E1 -30937.162,E2 -30937.162} C_VEL
LIN {X 0,Y 53.885,Z 268.315,A -85,B 0,C 180,E1 -30941.016,E2 -30941.016} C_VEL
LIN {X 0,Y 62.358,Z 259.599,A -85,B 0,C 180,E1 -30943.337,E2 -30943.337} C_VEL
LIN {X 0,Y 70.934,Z 248.845,A -85,B 0,C 180,E1 -30945.021,E2 -30945.021} C_VEL
LIN {X 0,Y 77.812,Z 238.103,A -85,B 0,C 180,E1 -30946.157,E2 -30946.157} C_VEL
LIN {X 0,Y 83.814,Z 226.086,A -85,B 0,C 180,E1 -30947.108,E2 -30947.108} C_VEL
LIN {X 0,Y 88.642,Z 213.169,A -85,B 0,C 180,E1 -30947.936,E2 -30947.936} C_VEL
LIN {X 0,Y 91.858,Z 200.585,A -85,B 0,C 180,E1 -30948.567,E2 -30948.567} C_VEL
LIN {X 0,Y 93.456,Z 190.821,A -85,B 0,C 180,E1 -30948.9,E2 -30948.9} C_VEL
LIN {X 0,Y 93.304,Z 189.105,A -85,B 0,C 180,E1 -30952.114,E2 -30952.114} C_VEL
LIN {X 0,Y 93.338,Z 188.894,A -85,B 0,C 180,E1 -30957.303,E2 -30957.303} C_VEL
LIN {X 0,Y 93.496,Z 190.591,A -85,B 0,C 180,E1 -30960.421,E2 -30960.421} C_VEL
LIN {X 0,Y 91.193,Z 204.103,A -85,B 0,C 180,E1 -30960.793,E2 -30960.793} C_VEL
LIN {X 0,Y 87.335,Z 217.626,A -85,B 0,C 180,E1 -30961.182,E2 -30961.182} C_VEL
LIN {X 0,Y 82.618,Z 229.403,A -85,B 0,C 180,E1 -30961.736,E2 -30961.736} C_VEL
LIN {X 0,Y 76.493,Z 240.943,A -85,B 0,C 180,E1 -30962.308,E2 -30962.308} C_VEL
LIN {X 0,Y 69.518,Z 251.472,A -85,B 0,C 180,E1 -30963.297,E2 -30963.297} C_VEL
LIN {X 0,Y 61.685,Z 261.073,A -85,B 0,C 180,E1 -30964.485,E2 -30964.485} C_VEL
LIN {X 0,Y 53.081,Z 269.894,A -85,B 0,C 180,E1 -30966.771,E2 -30966.771} C_VEL
LIN {X 0,Y 42.809,Z 278.369,A -85,B 0,C 180,E1 -30969.921,E2 -30969.921} C_VEL
LIN {X 0,Y 32.938,Z 285.25,A -85,B 0,C 180,E1 -30976.22,E2 -30976.22} C_VEL
LIN {X 0,Y 23.623,Z 290.71,A -85,B 0,C 180,E1 -30986.806,E2 -30986.806} C_VEL
LIN {X 0,Y 16.067,Z 294.971,A -85,B 0,C 180,E1 -31008.992,E2 -31008.992} C_VEL
LIN {X 0,Y 13.321,Z 298.131,A -85,B 0,C 180,E1 -31049.997,E2 -31049.997} C_VEL
LIN {X 0,Y 14.587,Z 299.611,A -85,B 0,C 180,E1 -31078.8,E2 -31078.8} C_VEL
LIN {X 0,Y 18.402,Z 300.644,A -85,B 0,C 180,E1 -31099.802,E2 -31099.802} C_VEL
LIN {X 0,Y 29.848,Z 301.513,A -85,B 0,C 180,E1 -31120.361,E2 -31120.361} C_VEL
LIN {X 0,Y 43.005,Z 300.892,A -85,B 0,C 180,E1 -31128.675,E2 -31128.675} C_VEL
LIN {X 0,Y 56.648,Z 298.658,A -85,B 0,C 180,E1 -31132.984,E2 -31132.984} C_VEL
LIN {X 0,Y 67.015,Z 295.932,A -85,B 0,C 180,E1 -31135.056,E2 -31135.056} C_VEL
LIN {X 0,Y 77.453,Z 292.218,A -85,B 0,C 180,E1 -31136.498,E2 -31136.498} C_VEL
LIN {X 0,Y 77.402,Z 292.2,A -85,B 0,C 180,E1 -31137.182,E2 -31137.182} C_VEL
LIN {X 0,Y 66.776,Z 295.802,A -85,B 0,C 180,E1 -31138.992,E2 -31138.992} C_VEL
LIN {X 0,Y 56.242,Z 298.355,A -85,B 0,C 180,E1 -31141.447,E2 -31141.447} C_VEL
LIN {X 0,Y 49.292,Z 299.535,A -85,B 0,C 180,E1 -31143.577,E2 -31143.577} C_VEL
LIN {X 0,Y 42.436,Z 300.261,A -85,B 0,C 180,E1 -31146.451,E2 -31146.451} C_VEL
LIN {X 0,Y 29.218,Z 300.503,A -85,B 0,C 180,E1 -31155.815,E2 -31155.815} C_VEL
LIN {X 0,Y 23.092,Z 300.039,A -85,B 0,C 180,E1 -31164.073,E2 -31164.073} C_VEL
LIN {X 0,Y 17.731,Z 299.131,A -85,B 0,C 180,E1 -31177.56,E2 -31177.56} C_VEL
LIN {X 0,Y 14.034,Z 297.816,A -85,B 0,C 180,E1 -31199.95,E2 -31199.95} C_VEL
LIN {X 0,Y 14.447,Z 295.103,A -85,B 0,C 180,E1 -31243.372,E2 -31243.372} C_VEL
LIN {X 0,Y 16.445,Z 293.734,A -85,B 0,C 180,E1 -31257.509,E2 -31257.509} C_VEL
LIN {X 0,Y 19.58,Z 291.747,A -85,B 0,C 180,E1 -31272.113,E2 -31272.113} C_VEL
LIN {X 0,Y 25.355,Z 288.088,A -85,B 0,C 180,E1 -31290.621,E2 -31290.621} C_VEL
LIN {X 0,Y 32.388,Z 283.754,A -85,B 0,C 180,E1 -31301.822,E2 -31301.822} C_VEL
LIN {X 0,Y 37.153,Z 280.692,A -85,B 0,C 180,E1 -31304.915,E2 -31304.915} C_VEL
LIN {X 0,Y 46.81,Z 273.668,A -85,B 0,C 180,E1 -31307.404,E2 -31307.404} C_VEL
LIN {X 0,Y 55.486,Z 266.03,A -85,B 0,C 180,E1 -31309.006,E2 -31309.006} C_VEL
LIN {X 0,Y 64.193,Z 256.738,A -85,B 0,C 180,E1 -31310.181,E2 -31310.181} C_VEL
LIN {X 0,Y 72.066,Z 246.366,A -85,B 0,C 180,E1 -31310.904,E2 -31310.904} C_VEL
LIN {X 0,Y 79.056,Z 234.868,A -85,B 0,C 180,E1 -31311.499,E2 -31311.499} C_VEL
LIN {X 0,Y 84.701,Z 222.861,A -85,B 0,C 180,E1 -31312.105,E2 -31312.105} C_VEL
LIN {X 0,Y 89.17,Z 209.808,A -85,B 0,C 180,E1 -31312.652,E2 -31312.652} C_VEL
LIN {X 0,Y 92.162,Z 196.724,A -85,B 0,C 180,E1 -31313.093,E2 -31313.093} C_VEL
LIN {X 0,Y 92.274,Z 196.025,A -85,B 0,C 180,E1 -31313.26,E2 -31313.26} C_VEL
LIN {X 0,Y 92.31,Z 195.82,A -85,B 0,C 180,E1 -31316.104,E2 -31316.104} C_VEL
LIN {X 0,Y 89.824,Z 207.625,A -85,B 0,C 180,E1 -31316.374,E2 -31316.374} C_VEL
LIN {X 0,Y 85.793,Z 220.204,A -85,B 0,C 180,E1 -31316.607,E2 -31316.607} C_VEL
LIN {X 0,Y 80.064,Z 233.14,A -85,B 0,C 180,E1 -31316.866,E2 -31316.866} C_VEL
LIN {X 0,Y 73.89,Z 243.877,A -85,B 0,C 180,E1 -31317.091,E2 -31317.091} C_VEL
LIN {X 0,Y 66.829,Z 253.768,A -85,B 0,C 180,E1 -31317.525,E2 -31317.525} C_VEL
LIN {X 0,Y 59.774,Z 261.975,A -85,B 0,C 180,E1 -31318.03,E2 -31318.03} C_VEL
LIN {X 0,Y 50.958,Z 270.526,A -85,B 0,C 180,E1 -31319.273,E2 -31319.273} C_VEL
LIN {X 0,Y 40.415,Z 278.805,A -85,B 0,C 180,E1 -31320.684,E2 -31320.684} C_VEL
LIN {X 0,Y 29.958,Z 285.537,A -85,B 0,C 180,E1 -31324.4,E2 -31324.4} C_VEL
LIN {X 0,Y 18.02,Z 291.625,A -85,B 0,C 180,E1 -31332.821,E2 -31332.821} C_VEL
LIN {X 0,Y 8.89,Z 295.574,A -85,B 0,C 180,E1 -31357.753,E2 -31357.753} C_VEL
LIN {X 0,Y 6.192,Z 297.591,A -85,B 0,C 180,E1 -31409.995,E2 -31409.995} C_VEL
LIN {X 0,Y 9.028,Z 299.1,A -85,B 0,C 180,E1 -31461.116,E2 -31461.116} C_VEL
LIN {X 0,Y 14.836,Z 300.183,A -85,B 0,C 180,E1 -31481.329,E2 -31481.329} C_VEL
LIN {X 0,Y 28.262,Z 301.113,A -85,B 0,C 180,E1 -31494.095,E2 -31494.095} C_VEL
LIN {X 0,Y 35.205,Z 301.022,A -85,B 0,C 180,E1 -31496.508,E2 -31496.508} C_VEL
LIN {X 0,Y 35.15,Z 300.955,A -85,B 0,C 180,E1 -31498.615,E2 -31498.615} C_VEL
LIN {X 0,Y 28.121,Z 300.909,A -85,B 0,C 180,E1 -31501.493,E2 -31501.493} C_VEL
LIN {X 0,Y 21.197,Z 300.477,A -85,B 0,C 180,E1 -31505.934,E2 -31505.934} C_VEL
LIN {X 0,Y 14.504,Z 299.624,A -85,B 0,C 180,E1 -31514.287,E2 -31514.287} C_VEL
LIN {X 0,Y 8.593,Z 298.337,A -85,B 0,C 180,E1 -31535.138,E2 -31535.138} C_VEL
LIN {X 0,Y 8.246,Z 295.382,A -85,B 0,C 180,E1 -31621.555,E2 -31621.555} C_VEL
LIN {X 0,Y 16.234,Z 291.951,A -85,B 0,C 180,E1 -31649.981,E2 -31649.981} C_VEL
LIN {X 0,Y 26.2,Z 287.172,A -85,B 0,C 180,E1 -31659.863,E2 -31659.863} C_VEL
LIN {X 0,Y 37.153,Z 280.692,A -85,B 0,C 180,E1 -31664.915,E2 -31664.915} C_VEL
LIN {X 0,Y 40.151,Z 282.382,A -85,B 0,C 180,E1 -31665.893,E2 -31665.893} C_VEL
LIN {X 0,Y 40.151,Z 600,A -85,B 0,C 180,E1 -31665.893,E2 -31665.893} C_VEL
LIN {X 0,Y 40.151,Z 600,A -85,B 0,C 180,E1 -31665.893,E2 -31665.893}

QRS_NEXT_CUT()

QRS_NEXT()
QRS_HOME()

END
